LIN {X 0,Y 353.397,Z 547.439,A -85,B 0,C 180,E1 -13404.296,E2 -13404.296} C_VEL
LIN {X 0,Y 353.36,Z 549.314,A -85,B 0,C 180,E1 -13405.439,E2 -13405.439} C_VEL
LIN {X 0,Y 353.319,Z 551.736,A -85,B 0,C 180,E1 -13407.722,E2 -13407.722} C_VEL
LIN {X 0,Y 353.4,Z 552.359,A -85,B 0,C 180,E1 -13408.863,E2 -13408.863} C_VEL
LIN {X 0,Y 353.411,Z 552.568,A -85,B 0,C 180,E1 -13410.002,E2 -13410.002} C_VEL
LIN {X 0,Y 353.421,Z 552.342,A -85,B 0,C 180,E1 -13411.142,E2 -13411.142} C_VEL
LIN {X 0,Y 353.333,Z 551.718,A -85,B 0,C 180,E1 -13412.282,E2 -13412.282} C_VEL
LIN {X 0,Y 353.284,Z 550.703,A -85,B 0,C 180,E1 -13413.424,E2 -13413.424} C_VEL
LIN {X 0,Y 353.361,Z 549.273,A -85,B 0,C 180,E1 -13414.565,E2 -13414.565} C_VEL
LIN {X 0,Y 353.448,Z 546.504,A -85,B 0,C 180,E1 -13416.169,E2 -13416.169} C_VEL
LIN {X 0,Y 353.656,Z 542.242,A -85,B 0,C 180,E1 -13417.998,E2 -13417.998} C_VEL
LIN {X 0,Y 354.205,Z 536.027,A -85,B 0,C 180,E1 -13420,E2 -13420} C_VEL
LIN {X 0,Y 354.806,Z 529.25,A -85,B 0,C 180,E1 -13421.716,E2 -13421.716} C_VEL
LIN {X 0,Y 355.835,Z 520.862,A -85,B 0,C 180,E1 -13423.421,E2 -13423.421} C_VEL
LIN {X 0,Y 356.841,Z 510.928,A -85,B 0,C 180,E1 -13425.028,E2 -13425.028} C_VEL
LIN {X 0,Y 357.899,Z 500.395,A -85,B 0,C 180,E1 -13426.398,E2 -13426.398} C_VEL
LIN {X 0,Y 359.074,Z 489.567,A -85,B 0,C 180,E1 -13427.515,E2 -13427.515} C_VEL
LIN {X 0,Y 359.665,Z 483.015,A -85,B 0,C 180,E1 -13428.073,E2 -13428.073} C_VEL
LIN {X 0,Y 358.36,Z 470.302,A -85,B 0,C 180,E1 -13429.064,E2 -13429.064} C_VEL
LIN {X 0,Y 356.589,Z 457.253,A -85,B 0,C 180,E1 -13429.846,E2 -13429.846} C_VEL
LIN {X 0,Y 354.382,Z 444.691,A -85,B 0,C 180,E1 -13430.404,E2 -13430.404} C_VEL
LIN {X 0,Y 354.887,Z 437.431,A -85,B 0,C 180,E1 -13433.864,E2 -13433.864} C_VEL
LIN {X 0,Y 355.469,Z 430.621,A -85,B 0,C 180,E1 -13437.164,E2 -13437.164} C_VEL
LIN {X 0,Y 356.132,Z 424.489,A -85,B 0,C 180,E1 -13440.223,E2 -13440.223} C_VEL
LIN {X 0,Y 356.859,Z 418.153,A -85,B 0,C 180,E1 -13443.467,E2 -13443.467} C_VEL
LIN {X 0,Y 357.34,Z 414.367,A -85,B 0,C 180,E1 -13445.466,E2 -13445.466} C_VEL
LIN {X 0,Y 357.336,Z 410.539,A -85,B 0,C 180,E1 -13447.57,E2 -13447.57} C_VEL
LIN {X 0,Y 356.459,Z 405.441,A -85,B 0,C 180,E1 -13450.591,E2 -13450.591} C_VEL
LIN {X 0,Y 355.582,Z 400.398,A -85,B 0,C 180,E1 -13453.772,E2 -13453.772} C_VEL
LIN {X 0,Y 354.823,Z 396.289,A -85,B 0,C 180,E1 -13456.533,E2 -13456.533} C_VEL
LIN {X 0,Y 354.822,Z 396.289,A -85,B 0,C 180,E1 -13460.667,E2 -13460.667} C_VEL
LIN {X 0,Y 354.828,Z 396.285,A -85,B 0,C 180,E1 -13464.301,E2 -13464.301} C_VEL
LIN {X 0,Y 354.793,Z 396.287,A -85,B 0,C 180,E1 -13467.667,E2 -13467.667} C_VEL
LIN {X 0,Y 354.853,Z 396.28,A -85,B 0,C 180,E1 -13471.619,E2 -13471.619} C_VEL
LIN {X 0,Y 354.906,Z 396.275,A -85,B 0,C 180,E1 -13474.173,E2 -13474.173} C_VEL
LIN {X 0,Y 354.841,Z 396.282,A -85,B 0,C 180,E1 -13477.894,E2 -13477.894} C_VEL
LIN {X 0,Y 354.929,Z 396.272,A -85,B 0,C 180,E1 -13481.892,E2 -13481.892} C_VEL
LIN {X 0,Y 354.949,Z 396.27,A -85,B 0,C 180,E1 -13485.982,E2 -13485.982} C_VEL
LIN {X 0,Y 354.984,Z 396.265,A -85,B 0,C 180,E1 -13489.736,E2 -13489.736} C_VEL
LIN {X 0,Y 355.13,Z 396.245,A -85,B 0,C 180,E1 -13493.181,E2 -13493.181} C_VEL
LIN {X 0,Y 355.249,Z 396.233,A -85,B 0,C 180,E1 -13497.732,E2 -13497.732} C_VEL
LIN {X 0,Y 355.381,Z 396.22,A -85,B 0,C 180,E1 -13500,E2 -13500} C_VEL
LIN {X 0,Y 355.249,Z 396.235,A -85,B 0,C 180,E1 -13502.268,E2 -13502.268} C_VEL
LIN {X 0,Y 355.143,Z 396.244,A -85,B 0,C 180,E1 -13506.819,E2 -13506.819} C_VEL
LIN {X 0,Y 355.022,Z 396.259,A -85,B 0,C 180,E1 -13509.112,E2 -13509.112} C_VEL
LIN {X 0,Y 354.927,Z 396.271,A -85,B 0,C 180,E1 -13512.581,E2 -13512.581} C_VEL
LIN {X 0,Y 354.896,Z 396.278,A -85,B 0,C 180,E1 -13516.096,E2 -13516.096} C_VEL
LIN {X 0,Y 354.908,Z 396.274,A -85,B 0,C 180,E1 -13518.472,E2 -13518.472} C_VEL
LIN {X 0,Y 354.841,Z 396.283,A -85,B 0,C 180,E1 -13522.106,E2 -13522.106} C_VEL
LIN {X 0,Y 354.905,Z 396.277,A -85,B 0,C 180,E1 -13525.827,E2 -13525.827} C_VEL
LIN {X 0,Y 354.824,Z 396.288,A -85,B 0,C 180,E1 -13529.681,E2 -13529.681} C_VEL
LIN {X 0,Y 354.813,Z 396.288,A -85,B 0,C 180,E1 -13533.701,E2 -13533.701} C_VEL
LIN {X 0,Y 354.803,Z 396.286,A -85,B 0,C 180,E1 -13536.459,E2 -13536.459} C_VEL
LIN {X 0,Y 354.83,Z 396.288,A -85,B 0,C 180,E1 -13539.423,E2 -13539.423} C_VEL
LIN {X 0,Y 354.794,Z 396.29,A -85,B 0,C 180,E1 -13542.866,E2 -13542.866} C_VEL
LIN {X 0,Y 354.786,Z 396.288,A -85,B 0,C 180,E1 -13546.105,E2 -13546.105} C_VEL
LIN {X 0,Y 354.794,Z 396.293,A -85,B 0,C 180,E1 -13549.178,E2 -13549.178} C_VEL
LIN {X 0,Y 354.813,Z 396.286,A -85,B 0,C 180,E1 -13552.401,E2 -13552.401} C_VEL
LIN {X 0,Y 354.818,Z 396.29,A -85,B 0,C 180,E1 -13554.94,E2 -13554.94} C_VEL
LIN {X 0,Y 354.799,Z 396.288,A -85,B 0,C 180,E1 -13558.404,E2 -13558.404} C_VEL
LIN {X 0,Y 354.852,Z 396.281,A -85,B 0,C 180,E1 -13561.617,E2 -13561.617} C_VEL
LIN {X 0,Y 354.905,Z 396.274,A -85,B 0,C 180,E1 -13564.171,E2 -13564.171} C_VEL
LIN {X 0,Y 354.84,Z 396.282,A -85,B 0,C 180,E1 -13567.892,E2 -13567.892} C_VEL
LIN {X 0,Y 354.927,Z 396.271,A -85,B 0,C 180,E1 -13571.89,E2 -13571.89} C_VEL
LIN {X 0,Y 354.932,Z 396.271,A -85,B 0,C 180,E1 -13575.989,E2 -13575.989} C_VEL
LIN {X 0,Y 354.671,Z 396.303,A -85,B 0,C 180,E1 -13579.725,E2 -13579.725} C_VEL
LIN {X 0,Y 354.46,Z 396.335,A -85,B 0,C 180,E1 -13582.02,E2 -13582.02} C_VEL
LIN {X 0,Y 354.473,Z 399.377,A -85,B 0,C 180,E1 -13585.449,E2 -13585.449} C_VEL
LIN {X 0,Y 353.943,Z 403.666,A -85,B 0,C 180,E1 -13589.998,E2 -13589.998} C_VEL
LIN {X 0,Y 354.03,Z 406.198,A -85,B 0,C 180,E1 -13592.771,E2 -13592.771} C_VEL
LIN {X 0,Y 358.141,Z 421.163,A -85,B 0,C 180,E1 -13593.644,E2 -13593.644} C_VEL
LIN {X 0,Y 360.649,Z 432.415,A -85,B 0,C 180,E1 -13594.468,E2 -13594.468} C_VEL
LIN {X 0,Y 360.823,Z 435.833,A -85,B 0,C 180,E1 -13594.731,E2 -13594.731} C_VEL
LIN {X 0,Y 359.959,Z 448.009,A -85,B 0,C 180,E1 -13595.741,E2 -13595.741} C_VEL
LIN {X 0,Y 359.07,Z 457.581,A -85,B 0,C 180,E1 -13596.742,E2 -13596.742} C_VEL
LIN {X 0,Y 358.047,Z 466.663,A -85,B 0,C 180,E1 -13597.895,E2 -13597.895} C_VEL
LIN {X 0,Y 356.935,Z 476.618,A -85,B 0,C 180,E1 -13599.462,E2 -13599.462} C_VEL
LIN {X 0,Y 355.973,Z 484.984,A -85,B 0,C 180,E1 -13601.096,E2 -13601.096} C_VEL
LIN {X 0,Y 355.188,Z 492.159,A -85,B 0,C 180,E1 -13602.859,E2 -13602.859} C_VEL
LIN {X 0,Y 354.426,Z 498.743,A -85,B 0,C 180,E1 -13604.936,E2 -13604.936} C_VEL
LIN {X 0,Y 353.984,Z 503.035,A -85,B 0,C 180,E1 -13606.729,E2 -13606.729} C_VEL
LIN {X 0,Y 353.596,Z 506.211,A -85,B 0,C 180,E1 -13608.54,E2 -13608.54} C_VEL
LIN {X 0,Y 353.329,Z 508.636,A -85,B 0,C 180,E1 -13610.793,E2 -13610.793} C_VEL
LIN {X 0,Y 353.29,Z 509.396,A -85,B 0,C 180,E1 -13612.205,E2 -13612.205} C_VEL
LIN {X 0,Y 353.302,Z 509.483,A -85,B 0,C 180,E1 -13613.788,E2 -13613.788} C_VEL
LIN {X 0,Y 353.448,Z 508.434,A -85,B 0,C 180,E1 -13615.938,E2 -13615.938} C_VEL
LIN {X 0,Y 353.619,Z 507.123,A -85,B 0,C 180,E1 -13617.198,E2 -13617.198} C_VEL
LIN {X 0,Y 354.028,Z 504.148,A -85,B 0,C 180,E1 -13619.136,E2 -13619.136} C_VEL
LIN {X 0,Y 354.494,Z 500.016,A -85,B 0,C 180,E1 -13621.025,E2 -13621.025} C_VEL
LIN {X 0,Y 355.202,Z 494.331,A -85,B 0,C 180,E1 -13622.961,E2 -13622.961} C_VEL
LIN {X 0,Y 356.14,Z 486.878,A -85,B 0,C 180,E1 -13624.906,E2 -13624.906} C_VEL
LIN {X 0,Y 357.147,Z 479.057,A -85,B 0,C 180,E1 -13626.528,E2 -13626.528} C_VEL
LIN {X 0,Y 358.209,Z 469.992,A -85,B 0,C 180,E1 -13628.041,E2 -13628.041} C_VEL
LIN {X 0,Y 359.381,Z 459.402,A -85,B 0,C 180,E1 -13629.458,E2 -13629.458} C_VEL
LIN {X 0,Y 360.469,Z 448.14,A -85,B 0,C 180,E1 -13630.656,E2 -13630.656} C_VEL
LIN {X 0,Y 361.473,Z 436.115,A -85,B 0,C 180,E1 -13631.64,E2 -13631.64} C_VEL
LIN {X 0,Y 359.964,Z 428.14,A -85,B 0,C 180,E1 -13632.29,E2 -13632.29} C_VEL
LIN {X 0,Y 359.337,Z 425.606,A -85,B 0,C 180,E1 -13632.478,E2 -13632.478} C_VEL
LIN {X 0,Y 357.891,Z 422.365,A -85,B 0,C 180,E1 -13632.757,E2 -13632.757} C_VEL
LIN {X 0,Y 353.991,Z 417.862,A -85,B 0,C 180,E1 -13633.242,E2 -13633.242} C_VEL
LIN {X 0,Y 348.982,Z 412.465,A -85,B 0,C 180,E1 -13633.805,E2 -13633.805} C_VEL
LIN {X 0,Y 347.7,Z 410.318,A -85,B 0,C 180,E1 -13633.969,E2 -13633.969} C_VEL
LIN {X 0,Y 346.987,Z 407.79,A -85,B 0,C 180,E1 -13634.13,E2 -13634.13} C_VEL
LIN {X 0,Y 347.06,Z 405.464,A -85,B 0,C 180,E1 -13636.798,E2 -13636.798} C_VEL
LIN {X 0,Y 347.154,Z 402.495,A -85,B 0,C 180,E1 -13640.286,E2 -13640.286} C_VEL
LIN {X 0,Y 347.282,Z 400.542,A -85,B 0,C 180,E1 -13642.619,E2 -13642.619} C_VEL
LIN {X 0,Y 347.414,Z 397.753,A -85,B 0,C 180,E1 -13646.032,E2 -13646.032} C_VEL
LIN {X 0,Y 347.48,Z 397.209,A -85,B 0,C 180,E1 -13646.901,E2 -13646.901} C_VEL
LIN {X 0,Y 347.703,Z 397.178,A -85,B 0,C 180,E1 -13649.648,E2 -13649.648} C_VEL
LIN {X 0,Y 347.832,Z 397.16,A -85,B 0,C 180,E1 -13652.744,E2 -13652.744} C_VEL
LIN {X 0,Y 347.8,Z 397.164,A -85,B 0,C 180,E1 -13656.163,E2 -13656.163} C_VEL
LIN {X 0,Y 347.825,Z 397.157,A -85,B 0,C 180,E1 -13659.91,E2 -13659.91} C_VEL
LIN {X 0,Y 347.848,Z 397.156,A -85,B 0,C 180,E1 -13662.358,E2 -13662.358} C_VEL
LIN {X 0,Y 347.878,Z 397.153,A -85,B 0,C 180,E1 -13665.97,E2 -13665.97} C_VEL
LIN {X 0,Y 347.914,Z 397.146,A -85,B 0,C 180,E1 -13669.525,E2 -13669.525} C_VEL
LIN {X 0,Y 348.055,Z 397.13,A -85,B 0,C 180,E1 -13671.874,E2 -13671.874} C_VEL
LIN {X 0,Y 348.053,Z 397.132,A -85,B 0,C 180,E1 -13674.206,E2 -13674.206} C_VEL
LIN {X 0,Y 348.19,Z 397.114,A -85,B 0,C 180,E1 -13677.687,E2 -13677.687} C_VEL
LIN {X 0,Y 348.349,Z 397.094,A -85,B 0,C 180,E1 -13680,E2 -13680} C_VEL
LIN {X 0,Y 348.197,Z 397.113,A -85,B 0,C 180,E1 -13682.314,E2 -13682.314} C_VEL
LIN {X 0,Y 348.086,Z 397.127,A -85,B 0,C 180,E1 -13686.958,E2 -13686.958} C_VEL
LIN {X 0,Y 347.95,Z 397.144,A -85,B 0,C 180,E1 -13689.299,E2 -13689.299} C_VEL
LIN {X 0,Y 347.874,Z 397.154,A -85,B 0,C 180,E1 -13692.84,E2 -13692.84} C_VEL
LIN {X 0,Y 347.821,Z 397.16,A -85,B 0,C 180,E1 -13696.432,E2 -13696.432} C_VEL
LIN {X 0,Y 347.845,Z 397.157,A -85,B 0,C 180,E1 -13698.861,E2 -13698.861} C_VEL
LIN {X 0,Y 347.823,Z 397.164,A -85,B 0,C 180,E1 -13702.576,E2 -13702.576} C_VEL
LIN {X 0,Y 347.815,Z 397.165,A -85,B 0,C 180,E1 -13706.394,E2 -13706.394} C_VEL
LIN {X 0,Y 347.733,Z 397.174,A -85,B 0,C 180,E1 -13710.35,E2 -13710.35} C_VEL
LIN {X 0,Y 347.733,Z 397.172,A -85,B 0,C 180,E1 -13714.046,E2 -13714.046} C_VEL
LIN {X 0,Y 347.749,Z 397.171,A -85,B 0,C 180,E1 -13717.323,E2 -13717.323} C_VEL
LIN {X 0,Y 347.78,Z 397.17,A -85,B 0,C 180,E1 -13720.291,E2 -13720.291} C_VEL
LIN {X 0,Y 347.785,Z 397.199,A -85,B 0,C 180,E1 -13722.215,E2 -13722.215} C_VEL
LIN {X 0,Y 348.524,Z 400.99,A -85,B 0,C 180,E1 -13725.112,E2 -13725.112} C_VEL
LIN {X 0,Y 349.547,Z 406.827,A -85,B 0,C 180,E1 -13729.167,E2 -13729.167} C_VEL
LIN {X 0,Y 350.336,Z 411.714,A -85,B 0,C 180,E1 -13732.28,E2 -13732.28} C_VEL
LIN {X 0,Y 350.474,Z 413.477,A -85,B 0,C 180,E1 -13733.333,E2 -13733.333} C_VEL
LIN {X 0,Y 350.004,Z 417.843,A -85,B 0,C 180,E1 -13735.793,E2 -13735.793} C_VEL
LIN {X 0,Y 349.083,Z 425.275,A -85,B 0,C 180,E1 -13739.783,E2 -13739.783} C_VEL
LIN {X 0,Y 348.248,Z 432.816,A -85,B 0,C 180,E1 -13743.645,E2 -13743.645} C_VEL
LIN {X 0,Y 347.565,Z 440.422,A -85,B 0,C 180,E1 -13747.409,E2 -13747.409} C_VEL
LIN {X 0,Y 347.348,Z 443.506,A -85,B 0,C 180,E1 -13748.917,E2 -13748.917} C_VEL
LIN {X 0,Y 349.982,Z 457.043,A -85,B 0,C 180,E1 -13749.582,E2 -13749.582} C_VEL
LIN {X 0,Y 351.593,Z 469.541,A -85,B 0,C 180,E1 -13750.376,E2 -13750.376} C_VEL
LIN {X 0,Y 352.839,Z 482.403,A -85,B 0,C 180,E1 -13751.419,E2 -13751.419} C_VEL
LIN {X 0,Y 352.669,Z 487.333,A -85,B 0,C 180,E1 -13751.861,E2 -13751.861} C_VEL
LIN {X 0,Y 351.401,Z 498.465,A -85,B 0,C 180,E1 -13752.995,E2 -13752.995} C_VEL
LIN {X 0,Y 350.256,Z 508.181,A -85,B 0,C 180,E1 -13754.236,E2 -13754.236} C_VEL
LIN {X 0,Y 349.213,Z 517.642,A -85,B 0,C 180,E1 -13755.73,E2 -13755.73} C_VEL
LIN {X 0,Y 348.167,Z 526.574,A -85,B 0,C 180,E1 -13757.47,E2 -13757.47} C_VEL
LIN {X 0,Y 347.381,Z 533.764,A -85,B 0,C 180,E1 -13759.217,E2 -13759.217} C_VEL
LIN {X 0,Y 346.733,Z 540.34,A -85,B 0,C 180,E1 -13761.259,E2 -13761.259} C_VEL
LIN {X 0,Y 346.437,Z 544.705,A -85,B 0,C 180,E1 -13763.011,E2 -13763.011} C_VEL
LIN {X 0,Y 346.337,Z 547.027,A -85,B 0,C 180,E1 -13764.179,E2 -13764.179} C_VEL
LIN {X 0,Y 346.274,Z 548.895,A -85,B 0,C 180,E1 -13765.346,E2 -13765.346} C_VEL
LIN {X 0,Y 346.224,Z 551.312,A -85,B 0,C 180,E1 -13767.676,E2 -13767.676} C_VEL
LIN {X 0,Y 346.321,Z 551.933,A -85,B 0,C 180,E1 -13768.839,E2 -13768.839} C_VEL
LIN {X 0,Y 346.35,Z 552.137,A -85,B 0,C 180,E1 -13770.002,E2 -13770.002} C_VEL
LIN {X 0,Y 346.34,Z 551.906,A -85,B 0,C 180,E1 -13771.165,E2 -13771.165} C_VEL
LIN {X 0,Y 346.207,Z 550.26,A -85,B 0,C 180,E1 -13773.494,E2 -13773.494} C_VEL
LIN {X 0,Y 346.275,Z 548.823,A -85,B 0,C 180,E1 -13774.659,E2 -13774.659} C_VEL
LIN {X 0,Y 346.345,Z 546.379,A -85,B 0,C 180,E1 -13776.117,E2 -13776.117} C_VEL
LIN {X 0,Y 346.594,Z 541.777,A -85,B 0,C 180,E1 -13778.162,E2 -13778.162} C_VEL
LIN {X 0,Y 347.174,Z 535.549,A -85,B 0,C 180,E1 -13780.205,E2 -13780.205} C_VEL
LIN {X 0,Y 347.818,Z 528.762,A -85,B 0,C 180,E1 -13781.955,E2 -13781.955} C_VEL
LIN {X 0,Y 348.859,Z 520.356,A -85,B 0,C 180,E1 -13783.695,E2 -13783.695} C_VEL
LIN {X 0,Y 349.897,Z 510.606,A -85,B 0,C 180,E1 -13785.303,E2 -13785.303} C_VEL
LIN {X 0,Y 351.08,Z 499.852,A -85,B 0,C 180,E1 -13786.726,E2 -13786.726} C_VEL
LIN {X 0,Y 352.28,Z 488.975,A -85,B 0,C 180,E1 -13787.864,E2 -13787.864} C_VEL
LIN {X 0,Y 352.66,Z 482.378,A -85,B 0,C 180,E1 -13788.445,E2 -13788.445} C_VEL
LIN {X 0,Y 351.429,Z 470.426,A -85,B 0,C 180,E1 -13789.398,E2 -13789.398} C_VEL
LIN {X 0,Y 349.705,Z 457.486,A -85,B 0,C 180,E1 -13790.204,E2 -13790.204} C_VEL
LIN {X 0,Y 347.371,Z 444.293,A -85,B 0,C 180,E1 -13790.815,E2 -13790.815} C_VEL
LIN {X 0,Y 347.93,Z 436.473,A -85,B 0,C 180,E1 -13794.635,E2 -13794.635} C_VEL
LIN {X 0,Y 348.646,Z 429.181,A -85,B 0,C 180,E1 -13798.277,E2 -13798.277} C_VEL
LIN {X 0,Y 349.334,Z 422.844,A -85,B 0,C 180,E1 -13801.541,E2 -13801.541} C_VEL
LIN {X 0,Y 350.155,Z 417.016,A -85,B 0,C 180,E1 -13804.622,E2 -13804.622} C_VEL
LIN {X 0,Y 350.457,Z 412.746,A -85,B 0,C 180,E1 -13806.987,E2 -13806.987} C_VEL
LIN {X 0,Y 349.634,Z 407.634,A -85,B 0,C 180,E1 -13810.035,E2 -13810.035} C_VEL
LIN {X 0,Y 348.707,Z 402.209,A -85,B 0,C 180,E1 -13813.484,E2 -13813.484} C_VEL
LIN {X 0,Y 347.757,Z 397.17,A -85,B 0,C 180,E1 -13816.974,E2 -13816.974} C_VEL
LIN {X 0,Y 347.754,Z 397.168,A -85,B 0,C 180,E1 -13820.174,E2 -13820.174} C_VEL
LIN {X 0,Y 347.768,Z 397.168,A -85,B 0,C 180,E1 -13822.68,E2 -13822.68} C_VEL
LIN {X 0,Y 347.755,Z 397.164,A -85,B 0,C 180,E1 -13825.957,E2 -13825.957} C_VEL
LIN {X 0,Y 347.756,Z 397.164,A -85,B 0,C 180,E1 -13829.653,E2 -13829.653} C_VEL
LIN {X 0,Y 347.838,Z 397.154,A -85,B 0,C 180,E1 -13833.608,E2 -13833.608} C_VEL
LIN {X 0,Y 347.796,Z 397.161,A -85,B 0,C 180,E1 -13836.162,E2 -13836.162} C_VEL
LIN {X 0,Y 347.819,Z 397.157,A -85,B 0,C 180,E1 -13839.91,E2 -13839.91} C_VEL
LIN {X 0,Y 347.873,Z 397.155,A -85,B 0,C 180,E1 -13842.359,E2 -13842.359} C_VEL
LIN {X 0,Y 347.905,Z 397.148,A -85,B 0,C 180,E1 -13845.971,E2 -13845.971} C_VEL
LIN {X 0,Y 347.935,Z 397.142,A -85,B 0,C 180,E1 -13849.526,E2 -13849.526} C_VEL
LIN {X 0,Y 348.097,Z 397.122,A -85,B 0,C 180,E1 -13853.042,E2 -13853.042} C_VEL
LIN {X 0,Y 348.211,Z 397.109,A -85,B 0,C 180,E1 -13857.686,E2 -13857.686} C_VEL
LIN {X 0,Y 348.331,Z 397.098,A -85,B 0,C 180,E1 -13860,E2 -13860} C_VEL
LIN {X 0,Y 348.211,Z 397.11,A -85,B 0,C 180,E1 -13862.313,E2 -13862.313} C_VEL
LIN {X 0,Y 348.111,Z 397.12,A -85,B 0,C 180,E1 -13866.957,E2 -13866.957} C_VEL
LIN {X 0,Y 347.935,Z 397.143,A -85,B 0,C 180,E1 -13870.474,E2 -13870.474} C_VEL
LIN {X 0,Y 347.905,Z 397.148,A -85,B 0,C 180,E1 -13874.15,E2 -13874.15} C_VEL
LIN {X 0,Y 347.897,Z 397.147,A -85,B 0,C 180,E1 -13878.29,E2 -13878.29} C_VEL
LIN {X 0,Y 347.795,Z 397.165,A -85,B 0,C 180,E1 -13881.634,E2 -13881.634} C_VEL
LIN {X 0,Y 347.819,Z 397.158,A -85,B 0,C 180,E1 -13885.108,E2 -13885.108} C_VEL
LIN {X 0,Y 347.815,Z 397.161,A -85,B 0,C 180,E1 -13887.693,E2 -13887.693} C_VEL
LIN {X 0,Y 347.755,Z 397.164,A -85,B 0,C 180,E1 -13890.347,E2 -13890.347} C_VEL
LIN {X 0,Y 347.755,Z 397.165,A -85,B 0,C 180,E1 -13894.043,E2 -13894.043} C_VEL
LIN {X 0,Y 347.767,Z 397.168,A -85,B 0,C 180,E1 -13897.32,E2 -13897.32} C_VEL
LIN {X 0,Y 347.738,Z 397.166,A -85,B 0,C 180,E1 -13900.296,E2 -13900.296} C_VEL
LIN {X 0,Y 347.729,Z 397.171,A -85,B 0,C 180,E1 -13903.407,E2 -13903.407} C_VEL
LIN {X 0,Y 347.734,Z 397.168,A -85,B 0,C 180,E1 -13906.685,E2 -13906.685} C_VEL
LIN {X 0,Y 347.753,Z 397.164,A -85,B 0,C 180,E1 -13910.172,E2 -13910.172} C_VEL
LIN {X 0,Y 347.768,Z 397.165,A -85,B 0,C 180,E1 -13912.678,E2 -13912.678} C_VEL
LIN {X 0,Y 347.754,Z 397.164,A -85,B 0,C 180,E1 -13915.955,E2 -13915.955} C_VEL
LIN {X 0,Y 347.755,Z 397.164,A -85,B 0,C 180,E1 -13919.651,E2 -13919.651} C_VEL
LIN {X 0,Y 347.836,Z 397.154,A -85,B 0,C 180,E1 -13923.606,E2 -13923.606} C_VEL
LIN {X 0,Y 347.794,Z 397.16,A -85,B 0,C 180,E1 -13926.16,E2 -13926.16} C_VEL
LIN {X 0,Y 347.817,Z 397.156,A -85,B 0,C 180,E1 -13929.908,E2 -13929.908} C_VEL
LIN {X 0,Y 347.871,Z 397.152,A -85,B 0,C 180,E1 -13932.358,E2 -13932.358} C_VEL
LIN {X 0,Y 347.901,Z 397.147,A -85,B 0,C 180,E1 -13935.969,E2 -13935.969} C_VEL
LIN {X 0,Y 347.657,Z 397.176,A -85,B 0,C 180,E1 -13939.515,E2 -13939.515} C_VEL
LIN {X 0,Y 347.434,Z 397.208,A -85,B 0,C 180,E1 -13941.858,E2 -13941.858} C_VEL
LIN {X 0,Y 347.44,Z 400.136,A -85,B 0,C 180,E1 -13945.357,E2 -13945.357} C_VEL
LIN {X 0,Y 346.885,Z 404.449,A -85,B 0,C 180,E1 -13949.998,E2 -13949.998} C_VEL
LIN {X 0,Y 346.935,Z 406.636,A -85,B 0,C 180,E1 -13952.356,E2 -13952.356} C_VEL
LIN {X 0,Y 351.006,Z 420.997,A -85,B 0,C 180,E1 -13953.226,E2 -13953.226} C_VEL
LIN {X 0,Y 353.758,Z 433.144,A -85,B 0,C 180,E1 -13954.135,E2 -13954.135} C_VEL
LIN {X 0,Y 354.051,Z 436.48,A -85,B 0,C 180,E1 -13954.405,E2 -13954.405} C_VEL
LIN {X 0,Y 353.176,Z 448.27,A -85,B 0,C 180,E1 -13955.4,E2 -13955.4} C_VEL
LIN {X 0,Y 352.234,Z 458.052,A -85,B 0,C 180,E1 -13956.442,E2 -13956.442} C_VEL
LIN {X 0,Y 351.079,Z 468.119,A -85,B 0,C 180,E1 -13957.763,E2 -13957.763} C_VEL
LIN {X 0,Y 350.004,Z 477.238,A -85,B 0,C 180,E1 -13959.242,E2 -13959.242} C_VEL
LIN {X 0,Y 349.113,Z 484.74,A -85,B 0,C 180,E1 -13960.729,E2 -13960.729} C_VEL
LIN {X 0,Y 348.247,Z 492.091,A -85,B 0,C 180,E1 -13962.527,E2 -13962.527} C_VEL
LIN {X 0,Y 347.632,Z 497.065,A -85,B 0,C 180,E1 -13964.038,E2 -13964.038} C_VEL
LIN {X 0,Y 347.116,Z 501.841,A -85,B 0,C 180,E1 -13965.86,E2 -13965.86} C_VEL
LIN {X 0,Y 346.685,Z 505.459,A -85,B 0,C 180,E1 -13967.7,E2 -13967.7} C_VEL
LIN {X 0,Y 346.46,Z 507.25,A -85,B 0,C 180,E1 -13968.936,E2 -13968.936} C_VEL
LIN {X 0,Y 346.253,Z 509.224,A -85,B 0,C 180,E1 -13970.985,E2 -13970.985} C_VEL
LIN {X 0,Y 346.185,Z 509.916,A -85,B 0,C 180,E1 -13972.686,E2 -13972.686} C_VEL
LIN {X 0,Y 346.227,Z 509.896,A -85,B 0,C 180,E1 -13974.014,E2 -13974.014} C_VEL
LIN {X 0,Y 346.273,Z 509.403,A -85,B 0,C 180,E1 -13975.225,E2 -13975.225} C_VEL
LIN {X 0,Y 346.488,Z 508.125,A -85,B 0,C 180,E1 -13976.814,E2 -13976.814} C_VEL
LIN {X 0,Y 346.794,Z 506.003,A -85,B 0,C 180,E1 -13978.437,E2 -13978.437} C_VEL
LIN {X 0,Y 347.23,Z 502.364,A -85,B 0,C 180,E1 -13980.395,E2 -13980.395} C_VEL
LIN {X 0,Y 347.922,Z 497.176,A -85,B 0,C 180,E1 -13982.407,E2 -13982.407} C_VEL
LIN {X 0,Y 348.827,Z 490.635,A -85,B 0,C 180,E1 -13984.338,E2 -13984.338} C_VEL
LIN {X 0,Y 349.7,Z 483.775,A -85,B 0,C 180,E1 -13985.956,E2 -13985.956} C_VEL
LIN {X 0,Y 350.874,Z 474.829,A -85,B 0,C 180,E1 -13987.652,E2 -13987.652} C_VEL
LIN {X 0,Y 352.049,Z 464.804,A -85,B 0,C 180,E1 -13989.166,E2 -13989.166} C_VEL
LIN {X 0,Y 353.255,Z 454.028,A -85,B 0,C 180,E1 -13990.468,E2 -13990.468} C_VEL
LIN {X 0,Y 354.332,Z 442.706,A -85,B 0,C 180,E1 -13991.541,E2 -13991.541} C_VEL
LIN {X 0,Y 354.748,Z 436.625,A -85,B 0,C 180,E1 -13992.021,E2 -13992.021} C_VEL
LIN {X 0,Y 352.006,Z 424.655,A -85,B 0,C 180,E1 -13993.01,E2 -13993.01} C_VEL
LIN {X 0,Y 348.401,Z 412.41,A -85,B 0,C 180,E1 -13993.847,E2 -13993.847} C_VEL
LIN {X 0,Y 347.7,Z 410.318,A -85,B 0,C 180,E1 -13993.969,E2 -13993.969} C_VEL
LIN {X 0,Y 346.554,Z 408.686,A -85,B 0,C 180,E1 -13994.208,E2 -13994.208} C_VEL
LIN {X 0,Y 344.636,Z 407.492,A -85,B 0,C 180,E1 -13994.816,E2 -13994.816} C_VEL
LIN {X 0,Y 342.19,Z 406.75,A -85,B 0,C 180,E1 -13996.035,E2 -13996.035} C_VEL
LIN {X 0,Y 340.594,Z 405.909,A -85,B 0,C 180,E1 -13997.496,E2 -13997.496} C_VEL
LIN {X 0,Y 340.059,Z 404.553,A -85,B 0,C 180,E1 -13998.976,E2 -13998.976} C_VEL
LIN {X 0,Y 340.227,Z 402.274,A -85,B 0,C 180,E1 -14001.712,E2 -14001.712} C_VEL
LIN {X 0,Y 340.321,Z 399.878,A -85,B 0,C 180,E1 -14004.674,E2 -14004.674} C_VEL
LIN {X 0,Y 340.392,Z 398.73,A -85,B 0,C 180,E1 -14006.119,E2 -14006.119} C_VEL
LIN {X 0,Y 340.539,Z 398.074,A -85,B 0,C 180,E1 -14007.789,E2 -14007.789} C_VEL
LIN {X 0,Y 340.709,Z 398.047,A -85,B 0,C 180,E1 -14010.326,E2 -14010.326} C_VEL
LIN {X 0,Y 340.786,Z 398.037,A -85,B 0,C 180,E1 -14013.018,E2 -14013.018} C_VEL
LIN {X 0,Y 340.774,Z 398.04,A -85,B 0,C 180,E1 -14016.93,E2 -14016.93} C_VEL
LIN {X 0,Y 340.788,Z 398.037,A -85,B 0,C 180,E1 -14020.733,E2 -14020.733} C_VEL
LIN {X 0,Y 340.768,Z 398.04,A -85,B 0,C 180,E1 -14023.218,E2 -14023.218} C_VEL
LIN {X 0,Y 340.828,Z 398.028,A -85,B 0,C 180,E1 -14026.89,E2 -14026.89} C_VEL
LIN {X 0,Y 340.911,Z 398.019,A -85,B 0,C 180,E1 -14030.507,E2 -14030.507} C_VEL
LIN {X 0,Y 341.059,Z 397.998,A -85,B 0,C 180,E1 -14032.898,E2 -14032.898} C_VEL
LIN {X 0,Y 341.152,Z 397.99,A -85,B 0,C 180,E1 -14037.639,E2 -14037.639} C_VEL
LIN {X 0,Y 341.298,Z 397.972,A -85,B 0,C 180,E1 -14040,E2 -14040} C_VEL
LIN {X 0,Y 341.159,Z 397.99,A -85,B 0,C 180,E1 -14042.361,E2 -14042.361} C_VEL
LIN {X 0,Y 341.056,Z 398.003,A -85,B 0,C 180,E1 -14047.102,E2 -14047.102} C_VEL
LIN {X 0,Y 340.856,Z 398.026,A -85,B 0,C 180,E1 -14050.694,E2 -14050.694} C_VEL
LIN {X 0,Y 340.844,Z 398.029,A -85,B 0,C 180,E1 -14054.326,E2 -14054.326} C_VEL
LIN {X 0,Y 340.821,Z 398.033,A -85,B 0,C 180,E1 -14058.469,E2 -14058.469} C_VEL
LIN {X 0,Y 340.795,Z 398.037,A -85,B 0,C 180,E1 -14061.883,E2 -14061.883} C_VEL
LIN {X 0,Y 340.76,Z 398.043,A -85,B 0,C 180,E1 -14065.666,E2 -14065.666} C_VEL
LIN {X 0,Y 340.712,Z 398.049,A -85,B 0,C 180,E1 -14068.322,E2 -14068.322} C_VEL
LIN {X 0,Y 340.682,Z 398.052,A -85,B 0,C 180,E1 -14071.047,E2 -14071.047} C_VEL
LIN {X 0,Y 340.704,Z 398.048,A -85,B 0,C 180,E1 -14075.281,E2 -14075.281} C_VEL
LIN {X 0,Y 340.704,Z 398.049,A -85,B 0,C 180,E1 -14078.39,E2 -14078.39} C_VEL
LIN {X 0,Y 340.752,Z 398.118,A -85,B 0,C 180,E1 -14081.689,E2 -14081.689} C_VEL
LIN {X 0,Y 341.417,Z 401.553,A -85,B 0,C 180,E1 -14084.418,E2 -14084.418} C_VEL
LIN {X 0,Y 342.163,Z 406.035,A -85,B 0,C 180,E1 -14087.684,E2 -14087.684} C_VEL
LIN {X 0,Y 343.07,Z 411.152,A -85,B 0,C 180,E1 -14091.12,E2 -14091.12} C_VEL
LIN {X 0,Y 343.439,Z 415.151,A -85,B 0,C 180,E1 -14093.602,E2 -14093.602} C_VEL
LIN {X 0,Y 342.834,Z 420.066,A -85,B 0,C 180,E1 -14096.397,E2 -14096.397} C_VEL
LIN {X 0,Y 341.85,Z 427.473,A -85,B 0,C 180,E1 -14100.438,E2 -14100.438} C_VEL
LIN {X 0,Y 341.045,Z 434.974,A -85,B 0,C 180,E1 -14104.361,E2 -14104.361} C_VEL
LIN {X 0,Y 340.345,Z 443.121,A -85,B 0,C 180,E1 -14108.437,E2 -14108.437} C_VEL
LIN {X 0,Y 343.055,Z 456.588,A -85,B 0,C 180,E1 -14109.124,E2 -14109.124} C_VEL
LIN {X 0,Y 344.721,Z 469.437,A -85,B 0,C 180,E1 -14109.97,E2 -14109.97} C_VEL
LIN {X 0,Y 345.88,Z 482.178,A -85,B 0,C 180,E1 -14111.031,E2 -14111.031} C_VEL
LIN {X 0,Y 345.929,Z 487.092,A -85,B 0,C 180,E1 -14111.494,E2 -14111.494} C_VEL
LIN {X 0,Y 344.572,Z 498.178,A -85,B 0,C 180,E1 -14112.647,E2 -14112.647} C_VEL
LIN {X 0,Y 343.349,Z 508.192,A -85,B 0,C 180,E1 -14113.962,E2 -14113.962} C_VEL
LIN {X 0,Y 342.314,Z 517.302,A -85,B 0,C 180,E1 -14115.436,E2 -14115.436} C_VEL
LIN {X 0,Y 341.183,Z 526.217,A -85,B 0,C 180,E1 -14117.209,E2 -14117.209} C_VEL
LIN {X 0,Y 340.342,Z 533.386,A -85,B 0,C 180,E1 -14118.991,E2 -14118.991} C_VEL
LIN {X 0,Y 339.696,Z 539.951,A -85,B 0,C 180,E1 -14121.076,E2 -14121.076} C_VEL
LIN {X 0,Y 339.363,Z 544.303,A -85,B 0,C 180,E1 -14122.865,E2 -14122.865} C_VEL
LIN {X 0,Y 339.257,Z 546.62,A -85,B 0,C 180,E1 -14124.057,E2 -14124.057} C_VEL
LIN {X 0,Y 339.193,Z 548.479,A -85,B 0,C 180,E1 -14125.248,E2 -14125.248} C_VEL
LIN {X 0,Y 339.13,Z 550.888,A -85,B 0,C 180,E1 -14127.627,E2 -14127.627} C_VEL
LIN {X 0,Y 339.227,Z 551.506,A -85,B 0,C 180,E1 -14128.815,E2 -14128.815} C_VEL
LIN {X 0,Y 339.29,Z 551.705,A -85,B 0,C 180,E1 -14130.002,E2 -14130.002} C_VEL
LIN {X 0,Y 339.26,Z 551.471,A -85,B 0,C 180,E1 -14131.189,E2 -14131.189} C_VEL
LIN {X 0,Y 339.132,Z 549.817,A -85,B 0,C 180,E1 -14133.567,E2 -14133.567} C_VEL
LIN {X 0,Y 339.194,Z 548.371,A -85,B 0,C 180,E1 -14134.756,E2 -14134.756} C_VEL
LIN {X 0,Y 339.3,Z 545.37,A -85,B 0,C 180,E1 -14136.543,E2 -14136.543} C_VEL
LIN {X 0,Y 339.549,Z 541.306,A -85,B 0,C 180,E1 -14138.333,E2 -14138.333} C_VEL
LIN {X 0,Y 340.146,Z 535.061,A -85,B 0,C 180,E1 -14140.418,E2 -14140.418} C_VEL
LIN {X 0,Y 340.848,Z 528.258,A -85,B 0,C 180,E1 -14142.203,E2 -14142.203} C_VEL
LIN {X 0,Y 341.89,Z 519.822,A -85,B 0,C 180,E1 -14143.979,E2 -14143.979} C_VEL
LIN {X 0,Y 342.894,Z 511.129,A -85,B 0,C 180,E1 -14145.455,E2 -14145.455} C_VEL
LIN {X 0,Y 344.107,Z 500.438,A -85,B 0,C 180,E1 -14146.922,E2 -14146.922} C_VEL
LIN {X 0,Y 345.333,Z 489.847,A -85,B 0,C 180,E1 -14148.083,E2 -14148.083} C_VEL
LIN {X 0,Y 345.78,Z 483.476,A -85,B 0,C 180,E1 -14148.672,E2 -14148.672} C_VEL
LIN {X 0,Y 344.506,Z 470.63,A -85,B 0,C 180,E1 -14149.738,E2 -14149.738} C_VEL
LIN {X 0,Y 342.772,Z 457.349,A -85,B 0,C 180,E1 -14150.595,E2 -14150.595} C_VEL
LIN {X 0,Y 340.358,Z 443.875,A -85,B 0,C 180,E1 -14151.242,E2 -14151.242} C_VEL
LIN {X 0,Y 340.899,Z 436.614,A -85,B 0,C 180,E1 -14154.891,E2 -14154.891} C_VEL
LIN {X 0,Y 341.569,Z 430.051,A -85,B 0,C 180,E1 -14158.247,E2 -14158.247} C_VEL
LIN {X 0,Y 342.291,Z 423.742,A -85,B 0,C 180,E1 -14161.574,E2 -14161.574} C_VEL
LIN {X 0,Y 343.208,Z 417.41,A -85,B 0,C 180,E1 -14165.005,E2 -14165.005} C_VEL
LIN {X 0,Y 343.46,Z 413.787,A -85,B 0,C 180,E1 -14167.057,E2 -14167.057} C_VEL
LIN {X 0,Y 342.491,Z 408.008,A -85,B 0,C 180,E1 -14170.602,E2 -14170.602} C_VEL
LIN {X 0,Y 341.62,Z 402.89,A -85,B 0,C 180,E1 -14173.942,E2 -14173.942} C_VEL
LIN {X 0,Y 340.724,Z 398.045,A -85,B 0,C 180,E1 -14177.342,E2 -14177.342} C_VEL
LIN {X 0,Y 340.706,Z 398.046,A -85,B 0,C 180,E1 -14180.248,E2 -14180.248} C_VEL
LIN {X 0,Y 340.717,Z 398.041,A -85,B 0,C 180,E1 -14183.56,E2 -14183.56} C_VEL
LIN {X 0,Y 340.699,Z 398.044,A -85,B 0,C 180,E1 -14186.154,E2 -14186.154} C_VEL
LIN {X 0,Y 340.748,Z 398.039,A -85,B 0,C 180,E1 -14190.33,E2 -14190.33} C_VEL
LIN {X 0,Y 340.81,Z 398.031,A -85,B 0,C 180,E1 -14193.02,E2 -14193.02} C_VEL
LIN {X 0,Y 340.763,Z 398.035,A -85,B 0,C 180,E1 -14195.639,E2 -14195.639} C_VEL
LIN {X 0,Y 340.752,Z 398.036,A -85,B 0,C 180,E1 -14199.474,E2 -14199.474} C_VEL
LIN {X 0,Y 340.865,Z 398.024,A -85,B 0,C 180,E1 -14201.984,E2 -14201.984} C_VEL
LIN {X 0,Y 340.877,Z 398.021,A -85,B 0,C 180,E1 -14205.705,E2 -14205.705} C_VEL
LIN {X 0,Y 340.877,Z 398.021,A -85,B 0,C 180,E1 -14209.306,E2 -14209.306} C_VEL
LIN {X 0,Y 341.065,Z 397.998,A -85,B 0,C 180,E1 -14212.898,E2 -14212.898} C_VEL
LIN {X 0,Y 341.173,Z 397.985,A -85,B 0,C 180,E1 -14217.639,E2 -14217.639} C_VEL
LIN {X 0,Y 341.282,Z 397.975,A -85,B 0,C 180,E1 -14220,E2 -14220} C_VEL
LIN {X 0,Y 341.173,Z 397.986,A -85,B 0,C 180,E1 -14222.361,E2 -14222.361} C_VEL
LIN {X 0,Y 341.081,Z 397.995,A -85,B 0,C 180,E1 -14227.102,E2 -14227.102} C_VEL
LIN {X 0,Y 340.877,Z 398.021,A -85,B 0,C 180,E1 -14230.694,E2 -14230.694} C_VEL
LIN {X 0,Y 340.87,Z 398.023,A -85,B 0,C 180,E1 -14234.324,E2 -14234.324} C_VEL
LIN {X 0,Y 340.844,Z 398.025,A -85,B 0,C 180,E1 -14238.466,E2 -14238.466} C_VEL
LIN {X 0,Y 340.761,Z 398.039,A -85,B 0,C 180,E1 -14241.856,E2 -14241.856} C_VEL
LIN {X 0,Y 340.779,Z 398.038,A -85,B 0,C 180,E1 -14245.664,E2 -14245.664} C_VEL
LIN {X 0,Y 340.735,Z 398.039,A -85,B 0,C 180,E1 -14248.32,E2 -14248.32} C_VEL
LIN {X 0,Y 340.704,Z 398.044,A -85,B 0,C 180,E1 -14251.044,E2 -14251.044} C_VEL
LIN {X 0,Y 340.724,Z 398.044,A -85,B 0,C 180,E1 -14255.278,E2 -14255.278} C_VEL
LIN {X 0,Y 340.716,Z 398.041,A -85,B 0,C 180,E1 -14258.385,E2 -14258.385} C_VEL
LIN {X 0,Y 340.705,Z 398.042,A -85,B 0,C 180,E1 -14262.044,E2 -14262.044} C_VEL
LIN {X 0,Y 340.69,Z 398.047,A -85,B 0,C 180,E1 -14265.46,E2 -14265.46} C_VEL
LIN {X 0,Y 340.692,Z 398.046,A -85,B 0,C 180,E1 -14268.689,E2 -14268.689} C_VEL
LIN {X 0,Y 340.739,Z 398.038,A -85,B 0,C 180,E1 -14271.771,E2 -14271.771} C_VEL
LIN {X 0,Y 340.729,Z 398.04,A -85,B 0,C 180,E1 -14275.594,E2 -14275.594} C_VEL
LIN {X 0,Y 340.703,Z 398.048,A -85,B 0,C 180,E1 -14278.954,E2 -14278.954} C_VEL
LIN {X 0,Y 340.809,Z 398.034,A -85,B 0,C 180,E1 -14283.018,E2 -14283.018} C_VEL
LIN {X 0,Y 340.761,Z 398.035,A -85,B 0,C 180,E1 -14285.637,E2 -14285.637} C_VEL
LIN {X 0,Y 340.757,Z 398.036,A -85,B 0,C 180,E1 -14289.473,E2 -14289.473} C_VEL
LIN {X 0,Y 340.862,Z 398.023,A -85,B 0,C 180,E1 -14291.982,E2 -14291.982} C_VEL
LIN {X 0,Y 340.856,Z 398.023,A -85,B 0,C 180,E1 -14295.715,E2 -14295.715} C_VEL
LIN {X 0,Y 340.635,Z 398.051,A -85,B 0,C 180,E1 -14299.297,E2 -14299.297} C_VEL
LIN {X 0,Y 340.416,Z 398.081,A -85,B 0,C 180,E1 -14301.689,E2 -14301.689} C_VEL
LIN {X 0,Y 340.365,Z 399.874,A -85,B 0,C 180,E1 -14304.072,E2 -14304.072} C_VEL
LIN {X 0,Y 340.409,Z 400.894,A -85,B 0,C 180,E1 -14305.261,E2 -14305.261} C_VEL
LIN {X 0,Y 339.829,Z 405.211,A -85,B 0,C 180,E1 -14309.998,E2 -14309.998} C_VEL
LIN {X 0,Y 339.881,Z 407.207,A -85,B 0,C 180,E1 -14311.96,E2 -14311.96} C_VEL
LIN {X 0,Y 343.555,Z 419.655,A -85,B 0,C 180,E1 -14312.71,E2 -14312.71} C_VEL
LIN {X 0,Y 346.417,Z 431.56,A -85,B 0,C 180,E1 -14313.601,E2 -14313.601} C_VEL
LIN {X 0,Y 347.312,Z 436.55,A -85,B 0,C 180,E1 -14314.025,E2 -14314.025} C_VEL
LIN {X 0,Y 346.443,Z 448.331,A -85,B 0,C 180,E1 -14315.032,E2 -14315.032} C_VEL
LIN {X 0,Y 345.263,Z 459.699,A -85,B 0,C 180,E1 -14316.279,E2 -14316.279} C_VEL
LIN {X 0,Y 344.121,Z 469.544,A -85,B 0,C 180,E1 -14317.626,E2 -14317.626} C_VEL
LIN {X 0,Y 343.008,Z 478.506,A -85,B 0,C 180,E1 -14319.134,E2 -14319.134} C_VEL
LIN {X 0,Y 342.088,Z 485.871,A -85,B 0,C 180,E1 -14320.653,E2 -14320.653} C_VEL
LIN {X 0,Y 341.192,Z 493.051,A -85,B 0,C 180,E1 -14322.488,E2 -14322.488} C_VEL
LIN {X 0,Y 340.46,Z 498.788,A -85,B 0,C 180,E1 -14324.34,E2 -14324.34} C_VEL
LIN {X 0,Y 339.966,Z 503.259,A -85,B 0,C 180,E1 -14326.203,E2 -14326.203} C_VEL
LIN {X 0,Y 339.533,Z 506.61,A -85,B 0,C 180,E1 -14328.086,E2 -14328.086} C_VEL
LIN {X 0,Y 339.323,Z 508.27,A -85,B 0,C 180,E1 -14329.35,E2 -14329.35} C_VEL
LIN {X 0,Y 339.169,Z 509.806,A -85,B 0,C 180,E1 -14331.179,E2 -14331.179} C_VEL
LIN {X 0,Y 339.104,Z 510.42,A -85,B 0,C 180,E1 -14333.187,E2 -14333.187} C_VEL
LIN {X 0,Y 339.157,Z 510.193,A -85,B 0,C 180,E1 -14334.481,E2 -14334.481} C_VEL
LIN {X 0,Y 339.242,Z 509.521,A -85,B 0,C 180,E1 -14335.785,E2 -14335.785} C_VEL
LIN {X 0,Y 339.453,Z 508.369,A -85,B 0,C 180,E1 -14337.093,E2 -14337.093} C_VEL
LIN {X 0,Y 339.875,Z 505.645,A -85,B 0,C 180,E1 -14339.071,E2 -14339.071} C_VEL
LIN {X 0,Y 340.388,Z 501.647,A -85,B 0,C 180,E1 -14341.073,E2 -14341.073} C_VEL
LIN {X 0,Y 341.14,Z 496.223,A -85,B 0,C 180,E1 -14343.085,E2 -14343.085} C_VEL
LIN {X 0,Y 342.144,Z 489.092,A -85,B 0,C 180,E1 -14345.107,E2 -14345.107} C_VEL
LIN {X 0,Y 343.167,Z 481.781,A -85,B 0,C 180,E1 -14346.748,E2 -14346.748} C_VEL
LIN {X 0,Y 344.279,Z 473.192,A -85,B 0,C 180,E1 -14348.317,E2 -14348.317} C_VEL
LIN {X 0,Y 345.539,Z 463.349,A -85,B 0,C 180,E1 -14349.771,E2 -14349.771} C_VEL
LIN {X 0,Y 346.695,Z 453.275,A -85,B 0,C 180,E1 -14350.962,E2 -14350.962} C_VEL
LIN {X 0,Y 347.79,Z 441.766,A -85,B 0,C 180,E1 -14352.046,E2 -14352.046} C_VEL
LIN {X 0,Y 347.906,Z 437.327,A -85,B 0,C 180,E1 -14352.413,E2 -14352.413} C_VEL
LIN {X 0,Y 345.144,Z 425.284,A -85,B 0,C 180,E1 -14353.44,E2 -14353.44} C_VEL
LIN {X 0,Y 341.405,Z 412.928,A -85,B 0,C 180,E1 -14354.32,E2 -14354.32} C_VEL
LIN {X 0,Y 339.984,Z 408.248,A -85,B 0,C 180,E1 -14354.611,E2 -14354.611} C_VEL
LIN {X 0,Y 340.06,Z 404.872,A -85,B 0,C 180,E1 -14358.598,E2 -14358.598} C_VEL
LIN {X 0,Y 340.059,Z 404.553,A -85,B 0,C 180,E1 -14358.976,E2 -14358.976} C_VEL
LIN {X 0,Y 339.429,Z 403.82,A -85,B 0,C 180,E1 -14359.958,E2 -14359.958} C_VEL
LIN {X 0,Y 336.673,Z 402.891,A -85,B 0,C 180,E1 -14361.564,E2 -14361.564} C_VEL
LIN {X 0,Y 334.335,Z 402.193,A -85,B 0,C 180,E1 -14362.866,E2 -14362.866} C_VEL
LIN {X 0,Y 333.34,Z 401.534,A -85,B 0,C 180,E1 -14363.869,E2 -14363.869} C_VEL
LIN {X 0,Y 333.264,Z 401.278,A -85,B 0,C 180,E1 -14364.208,E2 -14364.208} C_VEL
LIN {X 0,Y 333.441,Z 398.958,A -85,B 0,C 180,E1 -14367.461,E2 -14367.461} C_VEL
LIN {X 0,Y 333.631,Z 398.931,A -85,B 0,C 180,E1 -14369.725,E2 -14369.725} C_VEL
LIN {X 0,Y 333.722,Z 398.918,A -85,B 0,C 180,E1 -14372.399,E2 -14372.399} C_VEL
LIN {X 0,Y 333.743,Z 398.917,A -85,B 0,C 180,E1 -14375.092,E2 -14375.092} C_VEL
LIN {X 0,Y 333.707,Z 398.92,A -85,B 0,C 180,E1 -14379.021,E2 -14379.021} C_VEL
LIN {X 0,Y 333.777,Z 398.908,A -85,B 0,C 180,E1 -14381.589,E2 -14381.589} C_VEL
LIN {X 0,Y 333.789,Z 398.908,A -85,B 0,C 180,E1 -14385.576,E2 -14385.576} C_VEL
LIN {X 0,Y 333.818,Z 398.903,A -85,B 0,C 180,E1 -14389.078,E2 -14389.078} C_VEL
LIN {X 0,Y 334.008,Z 398.876,A -85,B 0,C 180,E1 -14392.747,E2 -14392.747} C_VEL
LIN {X 0,Y 333.799,Z 398.907,A -85,B 0,C 180,E1 -14395.169,E2 -14395.169} C_VEL
LIN {X 0,Y 334.089,Z 398.87,A -85,B 0,C 180,E1 -14397.589,E2 -14397.589} C_VEL
LIN {X 0,Y 334.248,Z 398.85,A -85,B 0,C 180,E1 -14400,E2 -14400} C_VEL
LIN {X 0,Y 334.121,Z 398.866,A -85,B 0,C 180,E1 -14402.411,E2 -14402.411} C_VEL
LIN {X 0,Y 334.006,Z 398.881,A -85,B 0,C 180,E1 -14407.253,E2 -14407.253} C_VEL
LIN {X 0,Y 333.818,Z 398.902,A -85,B 0,C 180,E1 -14410.923,E2 -14410.923} C_VEL
LIN {X 0,Y 333.79,Z 398.908,A -85,B 0,C 180,E1 -14414.635,E2 -14414.635} C_VEL
LIN {X 0,Y 333.78,Z 398.909,A -85,B 0,C 180,E1 -14418.657,E2 -14418.657} C_VEL
LIN {X 0,Y 333.731,Z 398.918,A -85,B 0,C 180,E1 -14422.276,E2 -14422.276} C_VEL
LIN {X 0,Y 333.72,Z 398.92,A -85,B 0,C 180,E1 -14426.248,E2 -14426.248} C_VEL
LIN {X 0,Y 333.674,Z 398.926,A -85,B 0,C 180,E1 -14428.976,E2 -14428.976} C_VEL
LIN {X 0,Y 333.628,Z 398.929,A -85,B 0,C 180,E1 -14432.589,E2 -14432.589} C_VEL
LIN {X 0,Y 333.662,Z 398.925,A -85,B 0,C 180,E1 -14436.141,E2 -14436.141} C_VEL
LIN {X 0,Y 333.671,Z 398.926,A -85,B 0,C 180,E1 -14439.189,E2 -14439.189} C_VEL
LIN {X 0,Y 333.685,Z 399.064,A -85,B 0,C 180,E1 -14441.162,E2 -14441.162} C_VEL
LIN {X 0,Y 334.481,Z 403.047,A -85,B 0,C 180,E1 -14444.411,E2 -14444.411} C_VEL
LIN {X 0,Y 335.258,Z 407.71,A -85,B 0,C 180,E1 -14447.874,E2 -14447.874} C_VEL
LIN {X 0,Y 336.096,Z 412.482,A -85,B 0,C 180,E1 -14451.151,E2 -14451.151} C_VEL
LIN {X 0,Y 336.434,Z 416.126,A -85,B 0,C 180,E1 -14453.466,E2 -14453.466} C_VEL
LIN {X 0,Y 335.823,Z 420.988,A -85,B 0,C 180,E1 -14456.313,E2 -14456.313} C_VEL
LIN {X 0,Y 334.806,Z 428.388,A -85,B 0,C 180,E1 -14460.446,E2 -14460.446} C_VEL
LIN {X 0,Y 333.974,Z 435.762,A -85,B 0,C 180,E1 -14464.383,E2 -14464.383} C_VEL
LIN {X 0,Y 333.342,Z 442.693,A -85,B 0,C 180,E1 -14467.93,E2 -14467.93} C_VEL
LIN {X 0,Y 336.143,Z 456.297,A -85,B 0,C 180,E1 -14468.652,E2 -14468.652} C_VEL
LIN {X 0,Y 337.755,Z 468.133,A -85,B 0,C 180,E1 -14469.45,E2 -14469.45} C_VEL
LIN {X 0,Y 338.769,Z 480.031,A -85,B 0,C 180,E1 -14470.44,E2 -14470.44} C_VEL
LIN {X 0,Y 339.176,Z 486.888,A -85,B 0,C 180,E1 -14471.112,E2 -14471.112} C_VEL
LIN {X 0,Y 337.804,Z 497.909,A -85,B 0,C 180,E1 -14472.288,E2 -14472.288} C_VEL
LIN {X 0,Y 336.451,Z 508.265,A -85,B 0,C 180,E1 -14473.686,E2 -14473.686} C_VEL
LIN {X 0,Y 335.421,Z 517.006,A -85,B 0,C 180,E1 -14475.138,E2 -14475.138} C_VEL
LIN {X 0,Y 334.229,Z 525.861,A -85,B 0,C 180,E1 -14476.938,E2 -14476.938} C_VEL
LIN {X 0,Y 333.319,Z 533.007,A -85,B 0,C 180,E1 -14478.756,E2 -14478.756} C_VEL
LIN {X 0,Y 332.641,Z 539.562,A -85,B 0,C 180,E1 -14480.885,E2 -14480.885} C_VEL
LIN {X 0,Y 332.289,Z 543.904,A -85,B 0,C 180,E1 -14482.712,E2 -14482.712} C_VEL
LIN {X 0,Y 332.18,Z 546.217,A -85,B 0,C 180,E1 -14483.93,E2 -14483.93} C_VEL
LIN {X 0,Y 332.115,Z 548.067,A -85,B 0,C 180,E1 -14485.147,E2 -14485.147} C_VEL
LIN {X 0,Y 332.057,Z 549.466,A -85,B 0,C 180,E1 -14486.362,E2 -14486.362} C_VEL
LIN {X 0,Y 332.133,Z 551.082,A -85,B 0,C 180,E1 -14488.79,E2 -14488.79} C_VEL
LIN {X 0,Y 332.213,Z 551.271,A -85,B 0,C 180,E1 -14490.002,E2 -14490.002} C_VEL
LIN {X 0,Y 332.167,Z 551.031,A -85,B 0,C 180,E1 -14491.215,E2 -14491.215} C_VEL
LIN {X 0,Y 332.058,Z 549.369,A -85,B 0,C 180,E1 -14493.643,E2 -14493.643} C_VEL
LIN {X 0,Y 332.116,Z 547.91,A -85,B 0,C 180,E1 -14494.858,E2 -14494.858} C_VEL
LIN {X 0,Y 332.221,Z 544.897,A -85,B 0,C 180,E1 -14496.684,E2 -14496.684} C_VEL
LIN {X 0,Y 332.495,Z 540.822,A -85,B 0,C 180,E1 -14498.511,E2 -14498.511} C_VEL
LIN {X 0,Y 333.125,Z 534.56,A -85,B 0,C 180,E1 -14500.64,E2 -14500.64} C_VEL
LIN {X 0,Y 333.885,Z 527.744,A -85,B 0,C 180,E1 -14502.462,E2 -14502.462} C_VEL
LIN {X 0,Y 334.955,Z 519.281,A -85,B 0,C 180,E1 -14504.275,E2 -14504.275} C_VEL
LIN {X 0,Y 335.998,Z 510.381,A -85,B 0,C 180,E1 -14505.809,E2 -14505.809} C_VEL
LIN {X 0,Y 337.271,Z 499.846,A -85,B 0,C 180,E1 -14507.276,E2 -14507.276} C_VEL
LIN {X 0,Y 338.588,Z 489.223,A -85,B 0,C 180,E1 -14508.456,E2 -14508.456} C_VEL
LIN {X 0,Y 338.892,Z 484.498,A -85,B 0,C 180,E1 -14508.909,E2 -14508.909} C_VEL
LIN {X 0,Y 337.808,Z 472.603,A -85,B 0,C 180,E1 -14509.957,E2 -14509.957} C_VEL
LIN {X 0,Y 336.13,Z 459.181,A -85,B 0,C 180,E1 -14510.883,E2 -14510.883} C_VEL
LIN {X 0,Y 333.781,Z 445.854,A -85,B 0,C 180,E1 -14511.581,E2 -14511.581} C_VEL
LIN {X 0,Y 333.334,Z 443.473,A -85,B 0,C 180,E1 -14511.687,E2 -14511.687} C_VEL
LIN {X 0,Y 334.002,Z 435.832,A -85,B 0,C 180,E1 -14515.624,E2 -14515.624} C_VEL
LIN {X 0,Y 334.797,Z 428.371,A -85,B 0,C 180,E1 -14519.56,E2 -14519.56} C_VEL
LIN {X 0,Y 335.811,Z 420.83,A -85,B 0,C 180,E1 -14523.693,E2 -14523.693} C_VEL
LIN {X 0,Y 336.34,Z 417.049,A -85,B 0,C 180,E1 -14525.81,E2 -14525.81} C_VEL
LIN {X 0,Y 336.367,Z 414.298,A -85,B 0,C 180,E1 -14527.442,E2 -14527.442} C_VEL
LIN {X 0,Y 335.4,Z 408.592,A -85,B 0,C 180,E1 -14531.031,E2 -14531.031} C_VEL
LIN {X 0,Y 334.539,Z 403.563,A -85,B 0,C 180,E1 -14534.416,E2 -14534.416} C_VEL
LIN {X 0,Y 333.686,Z 398.922,A -85,B 0,C 180,E1 -14537.829,E2 -14537.829} C_VEL
LIN {X 0,Y 333.659,Z 398.925,A -85,B 0,C 180,E1 -14541.203,E2 -14541.203} C_VEL
LIN {X 0,Y 333.683,Z 398.917,A -85,B 0,C 180,E1 -14543.862,E2 -14543.862} C_VEL
LIN {X 0,Y 333.65,Z 398.922,A -85,B 0,C 180,E1 -14547.414,E2 -14547.414} C_VEL
LIN {X 0,Y 333.697,Z 398.918,A -85,B 0,C 180,E1 -14551.026,E2 -14551.026} C_VEL
LIN {X 0,Y 333.742,Z 398.91,A -85,B 0,C 180,E1 -14553.754,E2 -14553.754} C_VEL
LIN {X 0,Y 333.727,Z 398.912,A -85,B 0,C 180,E1 -14557.914,E2 -14557.914} C_VEL
LIN {X 0,Y 333.801,Z 398.903,A -85,B 0,C 180,E1 -14561.59,E2 -14561.59} C_VEL
LIN {X 0,Y 333.816,Z 398.901,A -85,B 0,C 180,E1 -14565.577,E2 -14565.577} C_VEL
LIN {X 0,Y 333.84,Z 398.898,A -85,B 0,C 180,E1 -14569.078,E2 -14569.078} C_VEL
LIN {X 0,Y 334.012,Z 398.877,A -85,B 0,C 180,E1 -14572.747,E2 -14572.747} C_VEL
LIN {X 0,Y 333.812,Z 398.901,A -85,B 0,C 180,E1 -14575.169,E2 -14575.169} C_VEL
LIN {X 0,Y 334.11,Z 398.865,A -85,B 0,C 180,E1 -14577.589,E2 -14577.589} C_VEL
LIN {X 0,Y 334.233,Z 398.853,A -85,B 0,C 180,E1 -14580,E2 -14580} C_VEL
LIN {X 0,Y 334.11,Z 398.866,A -85,B 0,C 180,E1 -14582.411,E2 -14582.411} C_VEL
LIN {X 0,Y 334.031,Z 398.872,A -85,B 0,C 180,E1 -14587.252,E2 -14587.252} C_VEL
LIN {X 0,Y 333.84,Z 398.897,A -85,B 0,C 180,E1 -14590.922,E2 -14590.922} C_VEL
LIN {X 0,Y 333.815,Z 398.9,A -85,B 0,C 180,E1 -14594.634,E2 -14594.634} C_VEL
LIN {X 0,Y 333.803,Z 398.901,A -85,B 0,C 180,E1 -14598.654,E2 -14598.654} C_VEL
LIN {X 0,Y 333.699,Z 398.915,A -85,B 0,C 180,E1 -14602.278,E2 -14602.278} C_VEL
LIN {X 0,Y 333.741,Z 398.91,A -85,B 0,C 180,E1 -14606.246,E2 -14606.246} C_VEL
LIN {X 0,Y 333.696,Z 398.916,A -85,B 0,C 180,E1 -14608.973,E2 -14608.973} C_VEL
LIN {X 0,Y 333.65,Z 398.919,A -85,B 0,C 180,E1 -14612.586,E2 -14612.586} C_VEL
LIN {X 0,Y 333.682,Z 398.917,A -85,B 0,C 180,E1 -14616.138,E2 -14616.138} C_VEL
LIN {X 0,Y 333.653,Z 398.925,A -85,B 0,C 180,E1 -14619.191,E2 -14619.191} C_VEL
LIN {X 0,Y 333.638,Z 398.922,A -85,B 0,C 180,E1 -14622.499,E2 -14622.499} C_VEL
LIN {X 0,Y 333.628,Z 398.924,A -85,B 0,C 180,E1 -14625.958,E2 -14625.958} C_VEL
LIN {X 0,Y 333.653,Z 398.924,A -85,B 0,C 180,E1 -14629.314,E2 -14629.314} C_VEL
LIN {X 0,Y 333.671,Z 398.923,A -85,B 0,C 180,E1 -14633.167,E2 -14633.167} C_VEL
LIN {X 0,Y 333.68,Z 398.92,A -85,B 0,C 180,E1 -14635.34,E2 -14635.34} C_VEL
LIN {X 0,Y 333.696,Z 398.915,A -85,B 0,C 180,E1 -14639.636,E2 -14639.636} C_VEL
LIN {X 0,Y 333.745,Z 398.911,A -85,B 0,C 180,E1 -14642.399,E2 -14642.399} C_VEL
LIN {X 0,Y 333.732,Z 398.914,A -85,B 0,C 180,E1 -14645.089,E2 -14645.089} C_VEL
LIN {X 0,Y 333.69,Z 398.919,A -85,B 0,C 180,E1 -14649.018,E2 -14649.018} C_VEL
LIN {X 0,Y 333.798,Z 398.902,A -85,B 0,C 180,E1 -14651.588,E2 -14651.588} C_VEL
LIN {X 0,Y 333.812,Z 398.901,A -85,B 0,C 180,E1 -14655.575,E2 -14655.575} C_VEL
LIN {X 0,Y 333.603,Z 398.928,A -85,B 0,C 180,E1 -14659.068,E2 -14659.068} C_VEL
LIN {X 0,Y 333.397,Z 398.955,A -85,B 0,C 180,E1 -14661.512,E2 -14661.512} C_VEL
LIN {X 0,Y 333.3,Z 399.664,A -85,B 0,C 180,E1 -14662.729,E2 -14662.729} C_VEL
LIN {X 0,Y 333.378,Z 401.7,A -85,B 0,C 180,E1 -14665.161,E2 -14665.161} C_VEL
LIN {X 0,Y 332.774,Z 405.987,A -85,B 0,C 180,E1 -14669.998,E2 -14669.998} C_VEL
LIN {X 0,Y 332.754,Z 407.459,A -85,B 0,C 180,E1 -14671.51,E2 -14671.51} C_VEL
LIN {X 0,Y 336.818,Z 420.88,A -85,B 0,C 180,E1 -14672.352,E2 -14672.352} C_VEL
LIN {X 0,Y 339.713,Z 433.205,A -85,B 0,C 180,E1 -14673.311,E2 -14673.311} C_VEL
LIN {X 0,Y 340.473,Z 437.209,A -85,B 0,C 180,E1 -14673.671,E2 -14673.671} C_VEL
LIN {X 0,Y 339.753,Z 447.556,A -85,B 0,C 180,E1 -14674.57,E2 -14674.57} C_VEL
LIN {X 0,Y 338.64,Z 458.675,A -85,B 0,C 180,E1 -14675.773,E2 -14675.773} C_VEL
LIN {X 0,Y 337.356,Z 468.995,A -85,B 0,C 180,E1 -14677.178,E2 -14677.178} C_VEL
LIN {X 0,Y 336.227,Z 478.099,A -85,B 0,C 180,E1 -14678.714,E2 -14678.714} C_VEL
LIN {X 0,Y 335.184,Z 485.993,A -85,B 0,C 180,E1 -14680.347,E2 -14680.347} C_VEL
LIN {X 0,Y 334.272,Z 492.965,A -85,B 0,C 180,E1 -14682.134,E2 -14682.134} C_VEL
LIN {X 0,Y 333.434,Z 499.197,A -85,B 0,C 180,E1 -14684.171,E2 -14684.171} C_VEL
LIN {X 0,Y 332.961,Z 503.366,A -85,B 0,C 180,E1 -14685.923,E2 -14685.923} C_VEL
LIN {X 0,Y 332.491,Z 507,A -85,B 0,C 180,E1 -14687.976,E2 -14687.976} C_VEL
LIN {X 0,Y 332.173,Z 509.174,A -85,B 0,C 180,E1 -14689.784,E2 -14689.784} C_VEL
LIN {X 0,Y 332.085,Z 510.352,A -85,B 0,C 180,E1 -14691.38,E2 -14691.38} C_VEL
LIN {X 0,Y 332.038,Z 510.806,A -85,B 0,C 180,E1 -14693.71,E2 -14693.71} C_VEL
LIN {X 0,Y 332.108,Z 510.445,A -85,B 0,C 180,E1 -14695.036,E2 -14695.036} C_VEL
LIN {X 0,Y 332.416,Z 508.597,A -85,B 0,C 180,E1 -14697.38,E2 -14697.38} C_VEL
LIN {X 0,Y 332.79,Z 506.362,A -85,B 0,C 180,E1 -14699.057,E2 -14699.057} C_VEL
LIN {X 0,Y 333.319,Z 502.463,A -85,B 0,C 180,E1 -14701.1,E2 -14701.1} C_VEL
LIN {X 0,Y 334.098,Z 497.148,A -85,B 0,C 180,E1 -14703.153,E2 -14703.153} C_VEL
LIN {X 0,Y 335.125,Z 490.525,A -85,B 0,C 180,E1 -14705.127,E2 -14705.127} C_VEL
LIN {X 0,Y 336.23,Z 482.818,A -85,B 0,C 180,E1 -14706.934,E2 -14706.934} C_VEL
LIN {X 0,Y 337.49,Z 473.625,A -85,B 0,C 180,E1 -14708.658,E2 -14708.658} C_VEL
LIN {X 0,Y 338.7,Z 464.573,A -85,B 0,C 180,E1 -14710.03,E2 -14710.03} C_VEL
LIN {X 0,Y 339.871,Z 454.875,A -85,B 0,C 180,E1 -14711.229,E2 -14711.229} C_VEL
LIN {X 0,Y 341.05,Z 443.527,A -85,B 0,C 180,E1 -14712.343,E2 -14712.343} C_VEL
LIN {X 0,Y 341.27,Z 439.014,A -85,B 0,C 180,E1 -14712.73,E2 -14712.73} C_VEL
LIN {X 0,Y 338.536,Z 426.92,A -85,B 0,C 180,E1 -14713.808,E2 -14713.808} C_VEL
LIN {X 0,Y 334.968,Z 415.041,A -85,B 0,C 180,E1 -14714.705,E2 -14714.705} C_VEL
LIN {X 0,Y 332.925,Z 408.711,A -85,B 0,C 180,E1 -14715.128,E2 -14715.128} C_VEL
LIN {X 0,Y 333.048,Z 405.359,A -85,B 0,C 180,E1 -14719.144,E2 -14719.144} C_VEL
LIN {X 0,Y 333.203,Z 402.807,A -85,B 0,C 180,E1 -14722.289,E2 -14722.289} C_VEL
LIN {X 0,Y 333.264,Z 401.278,A -85,B 0,C 180,E1 -14724.208,E2 -14724.208} C_VEL
LIN {X 0,Y 332.635,Z 400.622,A -85,B 0,C 180,E1 -14725.211,E2 -14725.211} C_VEL
LIN {X 0,Y 329.906,Z 400.024,A -85,B 0,C 180,E1 -14726.855,E2 -14726.855} C_VEL
LIN {X 0,Y 327.599,Z 399.851,A -85,B 0,C 180,E1 -14728.189,E2 -14728.189} C_VEL
LIN {X 0,Y 326.627,Z 399.815,A -85,B 0,C 180,E1 -14729.22,E2 -14729.22} C_VEL
LIN {X 0,Y 326.557,Z 399.811,A -85,B 0,C 180,E1 -14729.568,E2 -14729.568} C_VEL
LIN {X 0,Y 326.666,Z 399.796,A -85,B 0,C 180,E1 -14733.141,E2 -14733.141} C_VEL
LIN {X 0,Y 326.68,Z 399.796,A -85,B 0,C 180,E1 -14737.217,E2 -14737.217} C_VEL
LIN {X 0,Y 326.726,Z 399.787,A -85,B 0,C 180,E1 -14741.176,E2 -14741.176} C_VEL
LIN {X 0,Y 326.744,Z 399.785,A -85,B 0,C 180,E1 -14745.432,E2 -14745.432} C_VEL
LIN {X 0,Y 326.754,Z 399.784,A -85,B 0,C 180,E1 -14748.838,E2 -14748.838} C_VEL
LIN {X 0,Y 326.962,Z 399.755,A -85,B 0,C 180,E1 -14752.59,E2 -14752.59} C_VEL
LIN {X 0,Y 326.765,Z 399.784,A -85,B 0,C 180,E1 -14755.065,E2 -14755.065} C_VEL
LIN {X 0,Y 327.03,Z 399.749,A -85,B 0,C 180,E1 -14757.537,E2 -14757.537} C_VEL
LIN {X 0,Y 327.199,Z 399.728,A -85,B 0,C 180,E1 -14760,E2 -14760} C_VEL
LIN {X 0,Y 327.058,Z 399.746,A -85,B 0,C 180,E1 -14762.463,E2 -14762.463} C_VEL
LIN {X 0,Y 326.977,Z 399.757,A -85,B 0,C 180,E1 -14766.17,E2 -14766.17} C_VEL
LIN {X 0,Y 326.896,Z 399.768,A -85,B 0,C 180,E1 -14768.656,E2 -14768.656} C_VEL
LIN {X 0,Y 326.719,Z 399.788,A -85,B 0,C 180,E1 -14772.422,E2 -14772.422} C_VEL
LIN {X 0,Y 326.736,Z 399.787,A -85,B 0,C 180,E1 -14774.959,E2 -14774.959} C_VEL
LIN {X 0,Y 326.746,Z 399.785,A -85,B 0,C 180,E1 -14778.855,E2 -14778.855} C_VEL
LIN {X 0,Y 326.68,Z 399.796,A -85,B 0,C 180,E1 -14782.783,E2 -14782.783} C_VEL
LIN {X 0,Y 326.667,Z 399.799,A -85,B 0,C 180,E1 -14786.859,E2 -14786.859} C_VEL
LIN {X 0,Y 326.618,Z 399.806,A -85,B 0,C 180,E1 -14790.611,E2 -14790.611} C_VEL
LIN {X 0,Y 326.592,Z 399.806,A -85,B 0,C 180,E1 -14794.021,E2 -14794.021} C_VEL
LIN {X 0,Y 326.615,Z 399.803,A -85,B 0,C 180,E1 -14797.241,E2 -14797.241} C_VEL
LIN {X 0,Y 326.626,Z 399.822,A -85,B 0,C 180,E1 -14800.452,E2 -14800.452} C_VEL
LIN {X 0,Y 327.27,Z 403.278,A -85,B 0,C 180,E1 -14803.408,E2 -14803.408} C_VEL
LIN {X 0,Y 328.037,Z 407.562,A -85,B 0,C 180,E1 -14806.755,E2 -14806.755} C_VEL
LIN {X 0,Y 328.9,Z 412.487,A -85,B 0,C 180,E1 -14810.287,E2 -14810.287} C_VEL
LIN {X 0,Y 329.354,Z 415.258,A -85,B 0,C 180,E1 -14812.142,E2 -14812.142} C_VEL
LIN {X 0,Y 329.322,Z 418.522,A -85,B 0,C 180,E1 -14814.189,E2 -14814.189} C_VEL
LIN {X 0,Y 328.4,Z 424.392,A -85,B 0,C 180,E1 -14817.658,E2 -14817.658} C_VEL
LIN {X 0,Y 327.594,Z 430.489,A -85,B 0,C 180,E1 -14821.107,E2 -14821.107} C_VEL
LIN {X 0,Y 326.868,Z 436.839,A -85,B 0,C 180,E1 -14824.562,E2 -14824.562} C_VEL
LIN {X 0,Y 326.34,Z 442.093,A -85,B 0,C 180,E1 -14827.359,E2 -14827.359} C_VEL
LIN {X 0,Y 329.511,Z 457.546,A -85,B 0,C 180,E1 -14828.262,E2 -14828.262} C_VEL
LIN {X 0,Y 331.179,Z 470.535,A -85,B 0,C 180,E1 -14829.2,E2 -14829.2} C_VEL
LIN {X 0,Y 332.054,Z 481.874,A -85,B 0,C 180,E1 -14830.209,E2 -14830.209} C_VEL
LIN {X 0,Y 332.268,Z 488.246,A -85,B 0,C 180,E1 -14830.865,E2 -14830.865} C_VEL
LIN {X 0,Y 330.698,Z 500.03,A -85,B 0,C 180,E1 -14832.215,E2 -14832.215} C_VEL
LIN {X 0,Y 329.395,Z 509.56,A -85,B 0,C 180,E1 -14833.581,E2 -14833.581} C_VEL
LIN {X 0,Y 328.293,Z 518.295,A -85,B 0,C 180,E1 -14835.117,E2 -14835.117} C_VEL
LIN {X 0,Y 327.094,Z 526.797,A -85,B 0,C 180,E1 -14836.964,E2 -14836.964} C_VEL
LIN {X 0,Y 326.187,Z 533.661,A -85,B 0,C 180,E1 -14838.821,E2 -14838.821} C_VEL
LIN {X 0,Y 325.605,Z 539.175,A -85,B 0,C 180,E1 -14840.686,E2 -14840.686} C_VEL
LIN {X 0,Y 325.215,Z 543.506,A -85,B 0,C 180,E1 -14842.553,E2 -14842.553} C_VEL
LIN {X 0,Y 325.102,Z 546.068,A -85,B 0,C 180,E1 -14843.947,E2 -14843.947} C_VEL
LIN {X 0,Y 324.986,Z 549.051,A -85,B 0,C 180,E1 -14846.283,E2 -14846.283} C_VEL
LIN {X 0,Y 325.04,Z 550.657,A -85,B 0,C 180,E1 -14848.763,E2 -14848.763} C_VEL
LIN {X 0,Y 325.138,Z 550.838,A -85,B 0,C 180,E1 -14850.002,E2 -14850.002} C_VEL
LIN {X 0,Y 325.073,Z 550.591,A -85,B 0,C 180,E1 -14851.241,E2 -14851.241} C_VEL
LIN {X 0,Y 324.987,Z 548.921,A -85,B 0,C 180,E1 -14853.722,E2 -14853.722} C_VEL
LIN {X 0,Y 325.085,Z 545.843,A -85,B 0,C 180,E1 -14856.025,E2 -14856.025} C_VEL
LIN {X 0,Y 325.304,Z 541.799,A -85,B 0,C 180,E1 -14858.075,E2 -14858.075} C_VEL
LIN {X 0,Y 325.805,Z 536.951,A -85,B 0,C 180,E1 -14859.939,E2 -14859.939} C_VEL
LIN {X 0,Y 326.435,Z 530.827,A -85,B 0,C 180,E1 -14861.804,E2 -14861.804} C_VEL
LIN {X 0,Y 327.493,Z 523.228,A -85,B 0,C 180,E1 -14863.656,E2 -14863.656} C_VEL
LIN {X 0,Y 328.656,Z 514.365,A -85,B 0,C 180,E1 -14865.387,E2 -14865.387} C_VEL
LIN {X 0,Y 329.715,Z 504.91,A -85,B 0,C 180,E1 -14866.885,E2 -14866.885} C_VEL
LIN {X 0,Y 331.116,Z 494.207,A -85,B 0,C 180,E1 -14868.247,E2 -14868.247} C_VEL
LIN {X 0,Y 332.005,Z 485.43,A -85,B 0,C 180,E1 -14869.156,E2 -14869.156} C_VEL
LIN {X 0,Y 330.93,Z 473.159,A -85,B 0,C 180,E1 -14870.29,E2 -14870.29} C_VEL
LIN {X 0,Y 329.399,Z 460.469,A -85,B 0,C 180,E1 -14871.207,E2 -14871.207} C_VEL
LIN {X 0,Y 327.006,Z 446.848,A -85,B 0,C 180,E1 -14871.969,E2 -14871.969} C_VEL
LIN {X 0,Y 326.314,Z 443.029,A -85,B 0,C 180,E1 -14872.163,E2 -14872.163} C_VEL
LIN {X 0,Y 327.038,Z 435.527,A -85,B 0,C 180,E1 -14876.141,E2 -14876.141} C_VEL
LIN {X 0,Y 327.911,Z 427.98,A -85,B 0,C 180,E1 -14880.245,E2 -14880.245} C_VEL
LIN {X 0,Y 328.785,Z 421.69,A -85,B 0,C 180,E1 -14883.766,E2 -14883.766} C_VEL
LIN {X 0,Y 329.396,Z 416.684,A -85,B 0,C 180,E1 -14886.687,E2 -14886.687} C_VEL
LIN {X 0,Y 328.978,Z 413.034,A -85,B 0,C 180,E1 -14888.966,E2 -14888.966} C_VEL
LIN {X 0,Y 328.111,Z 407.834,A -85,B 0,C 180,E1 -14892.387,E2 -14892.387} C_VEL
LIN {X 0,Y 327.388,Z 403.956,A -85,B 0,C 180,E1 -14895.108,E2 -14895.108} C_VEL
LIN {X 0,Y 326.656,Z 399.796,A -85,B 0,C 180,E1 -14898.268,E2 -14898.268} C_VEL
LIN {X 0,Y 326.63,Z 399.8,A -85,B 0,C 180,E1 -14901.392,E2 -14901.392} C_VEL
LIN {X 0,Y 326.627,Z 399.802,A -85,B 0,C 180,E1 -14904.852,E2 -14904.852} C_VEL
LIN {X 0,Y 326.615,Z 399.798,A -85,B 0,C 180,E1 -14907.456,E2 -14907.456} C_VEL
LIN {X 0,Y 326.655,Z 399.796,A -85,B 0,C 180,E1 -14910.34,E2 -14910.34} C_VEL
LIN {X 0,Y 326.697,Z 399.792,A -85,B 0,C 180,E1 -14914.517,E2 -14914.517} C_VEL
LIN {X 0,Y 326.653,Z 399.799,A -85,B 0,C 180,E1 -14918.546,E2 -14918.546} C_VEL
LIN {X 0,Y 326.752,Z 399.781,A -85,B 0,C 180,E1 -14921.178,E2 -14921.178} C_VEL
LIN {X 0,Y 326.771,Z 399.779,A -85,B 0,C 180,E1 -14925.433,E2 -14925.433} C_VEL
LIN {X 0,Y 326.777,Z 399.779,A -85,B 0,C 180,E1 -14928.839,E2 -14928.839} C_VEL
LIN {X 0,Y 326.965,Z 399.757,A -85,B 0,C 180,E1 -14932.59,E2 -14932.59} C_VEL
LIN {X 0,Y 326.779,Z 399.777,A -85,B 0,C 180,E1 -14935.065,E2 -14935.065} C_VEL
LIN {X 0,Y 327.051,Z 399.744,A -85,B 0,C 180,E1 -14937.537,E2 -14937.537} C_VEL
LIN {X 0,Y 327.185,Z 399.731,A -85,B 0,C 180,E1 -14940,E2 -14940} C_VEL
LIN {X 0,Y 327.051,Z 399.744,A -85,B 0,C 180,E1 -14942.463,E2 -14942.463} C_VEL
LIN {X 0,Y 326.974,Z 399.749,A -85,B 0,C 180,E1 -14946.701,E2 -14946.701} C_VEL
LIN {X 0,Y 326.821,Z 399.776,A -85,B 0,C 180,E1 -14949.906,E2 -14949.906} C_VEL
LIN {X 0,Y 326.766,Z 399.783,A -85,B 0,C 180,E1 -14953.685,E2 -14953.685} C_VEL
LIN {X 0,Y 326.706,Z 399.789,A -85,B 0,C 180,E1 -14957.527,E2 -14957.527} C_VEL
LIN {X 0,Y 326.669,Z 399.789,A -85,B 0,C 180,E1 -14960.134,E2 -14960.134} C_VEL
LIN {X 0,Y 326.659,Z 399.793,A -85,B 0,C 180,E1 -14964.128,E2 -14964.128} C_VEL
LIN {X 0,Y 326.689,Z 399.789,A -85,B 0,C 180,E1 -14966.857,E2 -14966.857} C_VEL
LIN {X 0,Y 326.641,Z 399.793,A -85,B 0,C 180,E1 -14970.609,E2 -14970.609} C_VEL
LIN {X 0,Y 326.613,Z 399.797,A -85,B 0,C 180,E1 -14974.019,E2 -14974.019} C_VEL
LIN {X 0,Y 326.634,Z 399.799,A -85,B 0,C 180,E1 -14977.238,E2 -14977.238} C_VEL
LIN {X 0,Y 326.584,Z 399.805,A -85,B 0,C 180,E1 -14981.13,E2 -14981.13} C_VEL
LIN {X 0,Y 326.561,Z 399.804,A -85,B 0,C 180,E1 -14984.747,E2 -14984.747} C_VEL
LIN {X 0,Y 326.583,Z 399.801,A -85,B 0,C 180,E1 -14988.153,E2 -14988.153} C_VEL
LIN {X 0,Y 326.604,Z 399.8,A -85,B 0,C 180,E1 -14991.387,E2 -14991.387} C_VEL
LIN {X 0,Y 326.625,Z 399.8,A -85,B 0,C 180,E1 -14994.85,E2 -14994.85} C_VEL
LIN {X 0,Y 326.613,Z 399.799,A -85,B 0,C 180,E1 -14997.454,E2 -14997.454} C_VEL
LIN {X 0,Y 326.653,Z 399.793,A -85,B 0,C 180,E1 -15000.338,E2 -15000.338} C_VEL
LIN {X 0,Y 326.695,Z 399.791,A -85,B 0,C 180,E1 -15004.515,E2 -15004.515} C_VEL
LIN {X 0,Y 326.653,Z 399.797,A -85,B 0,C 180,E1 -15008.544,E2 -15008.544} C_VEL
LIN {X 0,Y 326.749,Z 399.782,A -85,B 0,C 180,E1 -15011.176,E2 -15011.176} C_VEL
LIN {X 0,Y 326.767,Z 399.779,A -85,B 0,C 180,E1 -15015.431,E2 -15015.431} C_VEL
LIN {X 0,Y 326.582,Z 399.805,A -85,B 0,C 180,E1 -15018.83,E2 -15018.83} C_VEL
LIN {X 0,Y 326.363,Z 399.832,A -85,B 0,C 180,E1 -15021.328,E2 -15021.328} C_VEL
LIN {X 0,Y 326.283,Z 400.442,A -85,B 0,C 180,E1 -15022.572,E2 -15022.572} C_VEL
LIN {X 0,Y 326.349,Z 402.528,A -85,B 0,C 180,E1 -15025.056,E2 -15025.056} C_VEL
LIN {X 0,Y 325.726,Z 406.869,A -85,B 0,C 180,E1 -15029.998,E2 -15029.998} C_VEL
LIN {X 0,Y 325.707,Z 407.798,A -85,B 0,C 180,E1 -15031.041,E2 -15031.041} C_VEL
LIN {X 0,Y 329.949,Z 421.739,A -85,B 0,C 180,E1 -15031.955,E2 -15031.955} C_VEL
LIN {X 0,Y 332.967,Z 434.636,A -85,B 0,C 180,E1 -15032.999,E2 -15032.999} C_VEL
LIN {X 0,Y 333.718,Z 439.596,A -85,B 0,C 180,E1 -15033.451,E2 -15033.451} C_VEL
LIN {X 0,Y 332.662,Z 451.264,A -85,B 0,C 180,E1 -15034.542,E2 -15034.542} C_VEL
LIN {X 0,Y 331.437,Z 462.441,A -85,B 0,C 180,E1 -15035.866,E2 -15035.866} C_VEL
LIN {X 0,Y 330.165,Z 472.367,A -85,B 0,C 180,E1 -15037.335,E2 -15037.335} C_VEL
LIN {X 0,Y 328.997,Z 480.937,A -85,B 0,C 180,E1 -15038.907,E2 -15038.907} C_VEL
LIN {X 0,Y 327.857,Z 489.177,A -85,B 0,C 180,E1 -15040.777,E2 -15040.777} C_VEL
LIN {X 0,Y 327.072,Z 494.97,A -85,B 0,C 180,E1 -15042.406,E2 -15042.406} C_VEL
LIN {X 0,Y 326.347,Z 500.356,A -85,B 0,C 180,E1 -15044.282,E2 -15044.282} C_VEL
LIN {X 0,Y 325.81,Z 504.783,A -85,B 0,C 180,E1 -15046.283,E2 -15046.283} C_VEL
LIN {X 0,Y 325.381,Z 507.778,A -85,B 0,C 180,E1 -15048.127,E2 -15048.127} C_VEL
LIN {X 0,Y 325.046,Z 510.063,A -85,B 0,C 180,E1 -15050.236,E2 -15050.236} C_VEL
LIN {X 0,Y 324.988,Z 510.873,A -85,B 0,C 180,E1 -15051.582,E2 -15051.582} C_VEL
LIN {X 0,Y 324.929,Z 511.245,A -85,B 0,C 180,E1 -15052.91,E2 -15052.91} C_VEL
LIN {X 0,Y 324.999,Z 511.011,A -85,B 0,C 180,E1 -15054.737,E2 -15054.737} C_VEL
LIN {X 0,Y 325.255,Z 509.562,A -85,B 0,C 180,E1 -15056.982,E2 -15056.982} C_VEL
LIN {X 0,Y 325.704,Z 507.056,A -85,B 0,C 180,E1 -15059.042,E2 -15059.042} C_VEL
LIN {X 0,Y 326.251,Z 503.289,A -85,B 0,C 180,E1 -15061.128,E2 -15061.128} C_VEL
LIN {X 0,Y 327.16,Z 497.501,A -85,B 0,C 180,E1 -15063.427,E2 -15063.427} C_VEL
LIN {X 0,Y 328.184,Z 491.289,A -85,B 0,C 180,E1 -15065.32,E2 -15065.32} C_VEL
LIN {X 0,Y 329.243,Z 484.081,A -85,B 0,C 180,E1 -15067.083,E2 -15067.083} C_VEL
LIN {X 0,Y 330.575,Z 475.076,A -85,B 0,C 180,E1 -15068.838,E2 -15068.838} C_VEL
LIN {X 0,Y 331.9,Z 465.566,A -85,B 0,C 180,E1 -15070.333,E2 -15070.333} C_VEL
LIN {X 0,Y 333.191,Z 455.307,A -85,B 0,C 180,E1 -15071.634,E2 -15071.634} C_VEL
LIN {X 0,Y 334.393,Z 444.242,A -85,B 0,C 180,E1 -15072.744,E2 -15072.744} C_VEL
LIN {X 0,Y 334.551,Z 440.246,A -85,B 0,C 180,E1 -15073.103,E2 -15073.103} C_VEL
LIN {X 0,Y 332.019,Z 428.893,A -85,B 0,C 180,E1 -15074.167,E2 -15074.167} C_VEL
LIN {X 0,Y 328.454,Z 416.734,A -85,B 0,C 180,E1 -15075.133,E2 -15075.133} C_VEL
LIN {X 0,Y 325.903,Z 409.176,A -85,B 0,C 180,E1 -15075.664,E2 -15075.664} C_VEL
LIN {X 0,Y 326.022,Z 405.881,A -85,B 0,C 180,E1 -15079.706,E2 -15079.706} C_VEL
LIN {X 0,Y 326.195,Z 403.336,A -85,B 0,C 180,E1 -15082.896,E2 -15082.896} C_VEL
LIN {X 0,Y 326.332,Z 400.984,A -85,B 0,C 180,E1 -15085.948,E2 -15085.948} C_VEL
LIN {X 0,Y 326.409,Z 399.864,A -85,B 0,C 180,E1 -15087.433,E2 -15087.433} C_VEL
LIN {X 0,Y 326.557,Z 399.811,A -85,B 0,C 180,E1 -15089.568,E2 -15089.568} C_VEL
LIN {X 0,Y 325.919,Z 399.89,A -85,B 0,C 180,E1 -15090.598,E2 -15090.598} C_VEL
LIN {X 0,Y 323.099,Z 400.24,A -85,B 0,C 180,E1 -15092.274,E2 -15092.274} C_VEL
LIN {X 0,Y 320.702,Z 400.54,A -85,B 0,C 180,E1 -15093.631,E2 -15093.631} C_VEL
LIN {X 0,Y 319.682,Z 400.666,A -85,B 0,C 180,E1 -15094.682,E2 -15094.682} C_VEL
LIN {X 0,Y 319.605,Z 400.676,A -85,B 0,C 180,E1 -15095.038,E2 -15095.038} C_VEL
LIN {X 0,Y 319.635,Z 400.671,A -85,B 0,C 180,E1 -15098.051,E2 -15098.051} C_VEL
LIN {X 0,Y 319.688,Z 400.664,A -85,B 0,C 180,E1 -15100.952,E2 -15100.952} C_VEL
LIN {X 0,Y 319.712,Z 400.661,A -85,B 0,C 180,E1 -15105.275,E2 -15105.275} C_VEL
LIN {X 0,Y 319.741,Z 400.654,A -85,B 0,C 180,E1 -15109.872,E2 -15109.872} C_VEL
LIN {X 0,Y 319.915,Z 400.633,A -85,B 0,C 180,E1 -15112.426,E2 -15112.426} C_VEL
LIN {X 0,Y 319.734,Z 400.659,A -85,B 0,C 180,E1 -15114.956,E2 -15114.956} C_VEL
LIN {X 0,Y 319.974,Z 400.628,A -85,B 0,C 180,E1 -15117.482,E2 -15117.482} C_VEL
LIN {X 0,Y 320.15,Z 400.606,A -85,B 0,C 180,E1 -15120,E2 -15120} C_VEL
LIN {X 0,Y 319.999,Z 400.625,A -85,B 0,C 180,E1 -15122.518,E2 -15122.518} C_VEL
LIN {X 0,Y 319.933,Z 400.635,A -85,B 0,C 180,E1 -15126.306,E2 -15126.306} C_VEL
LIN {X 0,Y 319.824,Z 400.648,A -85,B 0,C 180,E1 -15128.849,E2 -15128.849} C_VEL
LIN {X 0,Y 319.666,Z 400.667,A -85,B 0,C 180,E1 -15132.701,E2 -15132.701} C_VEL
LIN {X 0,Y 319.681,Z 400.666,A -85,B 0,C 180,E1 -15135.297,E2 -15135.297} C_VEL
LIN {X 0,Y 319.674,Z 400.667,A -85,B 0,C 180,E1 -15139.255,E2 -15139.255} C_VEL
LIN {X 0,Y 319.628,Z 400.674,A -85,B 0,C 180,E1 -15143.315,E2 -15143.315} C_VEL
LIN {X 0,Y 319.619,Z 400.677,A -85,B 0,C 180,E1 -15146.09,E2 -15146.09} C_VEL
LIN {X 0,Y 319.564,Z 400.684,A -85,B 0,C 180,E1 -15148.936,E2 -15148.936} C_VEL
LIN {X 0,Y 319.515,Z 400.69,A -85,B 0,C 180,E1 -15151.864,E2 -15151.864} C_VEL
LIN {X 0,Y 319.565,Z 400.681,A -85,B 0,C 180,E1 -15155.545,E2 -15155.545} C_VEL
LIN {X 0,Y 319.586,Z 400.678,A -85,B 0,C 180,E1 -15158.006,E2 -15158.006} C_VEL
LIN {X 0,Y 319.576,Z 400.698,A -85,B 0,C 180,E1 -15159.809,E2 -15159.809} C_VEL
LIN {X 0,Y 320.388,Z 405.04,A -85,B 0,C 180,E1 -15163.629,E2 -15163.629} C_VEL
LIN {X 0,Y 321.195,Z 409.688,A -85,B 0,C 180,E1 -15167.293,E2 -15167.293} C_VEL
LIN {X 0,Y 322.043,Z 414.446,A -85,B 0,C 180,E1 -15170.742,E2 -15170.742} C_VEL
LIN {X 0,Y 322.428,Z 418.013,A -85,B 0,C 180,E1 -15173.151,E2 -15173.151} C_VEL
LIN {X 0,Y 321.833,Z 422.75,A -85,B 0,C 180,E1 -15176.081,E2 -15176.081} C_VEL
LIN {X 0,Y 320.693,Z 430.24,A -85,B 0,C 180,E1 -15180.46,E2 -15180.46} C_VEL
LIN {X 0,Y 319.856,Z 437.022,A -85,B 0,C 180,E1 -15184.273,E2 -15184.273} C_VEL
LIN {X 0,Y 319.342,Z 441.897,A -85,B 0,C 180,E1 -15186.828,E2 -15186.828} C_VEL
LIN {X 0,Y 322.282,Z 455.384,A -85,B 0,C 180,E1 -15187.613,E2 -15187.613} C_VEL
LIN {X 0,Y 324.027,Z 467.245,A -85,B 0,C 180,E1 -15188.473,E2 -15188.473} C_VEL
LIN {X 0,Y 325.11,Z 480.071,A -85,B 0,C 180,E1 -15189.612,E2 -15189.612} C_VEL
LIN {X 0,Y 325.546,Z 488.051,A -85,B 0,C 180,E1 -15190.454,E2 -15190.454} C_VEL
LIN {X 0,Y 323.927,Z 499.79,A -85,B 0,C 180,E1 -15191.83,E2 -15191.83} C_VEL
LIN {X 0,Y 322.553,Z 509.286,A -85,B 0,C 180,E1 -15193.223,E2 -15193.223} C_VEL
LIN {X 0,Y 321.422,Z 517.992,A -85,B 0,C 180,E1 -15194.791,E2 -15194.791} C_VEL
LIN {X 0,Y 320.147,Z 526.462,A -85,B 0,C 180,E1 -15196.676,E2 -15196.676} C_VEL
LIN {X 0,Y 319.162,Z 533.306,A -85,B 0,C 180,E1 -15198.572,E2 -15198.572} C_VEL
LIN {X 0,Y 318.568,Z 538.804,A -85,B 0,C 180,E1 -15200.479,E2 -15200.479} C_VEL
LIN {X 0,Y 318.165,Z 543.119,A -85,B 0,C 180,E1 -15202.386,E2 -15202.386} C_VEL
LIN {X 0,Y 318.01,Z 545.927,A -85,B 0,C 180,E1 -15203.99,E2 -15203.99} C_VEL
LIN {X 0,Y 317.915,Z 548.638,A -85,B 0,C 180,E1 -15206.2,E2 -15206.2} C_VEL
LIN {X 0,Y 317.946,Z 550.232,A -85,B 0,C 180,E1 -15208.736,E2 -15208.736} C_VEL
LIN {X 0,Y 318.049,Z 550.403,A -85,B 0,C 180,E1 -15210.002,E2 -15210.002} C_VEL
LIN {X 0,Y 317.979,Z 550.152,A -85,B 0,C 180,E1 -15211.269,E2 -15211.269} C_VEL
LIN {X 0,Y 317.916,Z 548.472,A -85,B 0,C 180,E1 -15213.805,E2 -15213.805} C_VEL
LIN {X 0,Y 318.002,Z 545.648,A -85,B 0,C 180,E1 -15215.998,E2 -15215.998} C_VEL
LIN {X 0,Y 318.244,Z 541.315,A -85,B 0,C 180,E1 -15218.255,E2 -15218.255} C_VEL
LIN {X 0,Y 318.759,Z 536.45,A -85,B 0,C 180,E1 -15220.161,E2 -15220.161} C_VEL
LIN {X 0,Y 319.451,Z 530.307,A -85,B 0,C 180,E1 -15222.066,E2 -15222.066} C_VEL
LIN {X 0,Y 320.542,Z 522.683,A -85,B 0,C 180,E1 -15223.958,E2 -15223.958} C_VEL
LIN {X 0,Y 321.726,Z 514.158,A -85,B 0,C 180,E1 -15225.658,E2 -15225.658} C_VEL
LIN {X 0,Y 322.865,Z 504.285,A -85,B 0,C 180,E1 -15227.255,E2 -15227.255} C_VEL
LIN {X 0,Y 324.341,Z 493.538,A -85,B 0,C 180,E1 -15228.642,E2 -15228.642} C_VEL
LIN {X 0,Y 325.09,Z 486.289,A -85,B 0,C 180,E1 -15229.416,E2 -15229.416} C_VEL
LIN {X 0,Y 324.034,Z 473.555,A -85,B 0,C 180,E1 -15230.641,E2 -15230.641} C_VEL
LIN {X 0,Y 322.55,Z 460.854,A -85,B 0,C 180,E1 -15231.603,E2 -15231.603} C_VEL
LIN {X 0,Y 320.15,Z 447.124,A -85,B 0,C 180,E1 -15232.405,E2 -15232.405} C_VEL
LIN {X 0,Y 319.295,Z 442.68,A -85,B 0,C 180,E1 -15232.612,E2 -15232.612} C_VEL
LIN {X 0,Y 320.08,Z 435.076,A -85,B 0,C 180,E1 -15236.753,E2 -15236.753} C_VEL
LIN {X 0,Y 320.84,Z 428.793,A -85,B 0,C 180,E1 -15240.255,E2 -15240.255} C_VEL
LIN {X 0,Y 321.784,Z 422.446,A -85,B 0,C 180,E1 -15243.906,E2 -15243.906} C_VEL
LIN {X 0,Y 322.334,Z 418.525,A -85,B 0,C 180,E1 -15246.222,E2 -15246.222} C_VEL
LIN {X 0,Y 322.182,Z 415.301,A -85,B 0,C 180,E1 -15248.252,E2 -15248.252} C_VEL
LIN {X 0,Y 321.23,Z 409.774,A -85,B 0,C 180,E1 -15251.938,E2 -15251.938} C_VEL
LIN {X 0,Y 320.342,Z 404.911,A -85,B 0,C 180,E1 -15255.408,E2 -15255.408} C_VEL
LIN {X 0,Y 319.565,Z 400.681,A -85,B 0,C 180,E1 -15258.717,E2 -15258.717} C_VEL
LIN {X 0,Y 319.568,Z 400.679,A -85,B 0,C 180,E1 -15262.349,E2 -15262.349} C_VEL
LIN {X 0,Y 319.567,Z 400.679,A -85,B 0,C 180,E1 -15265.124,E2 -15265.124} C_VEL
LIN {X 0,Y 319.574,Z 400.678,A -85,B 0,C 180,E1 -15269.06,E2 -15269.06} C_VEL
LIN {X 0,Y 319.613,Z 400.675,A -85,B 0,C 180,E1 -15272.498,E2 -15272.498} C_VEL
LIN {X 0,Y 319.612,Z 400.67,A -85,B 0,C 180,E1 -15275.304,E2 -15275.304} C_VEL
LIN {X 0,Y 319.604,Z 400.673,A -85,B 0,C 180,E1 -15278.048,E2 -15278.048} C_VEL
LIN {X 0,Y 319.697,Z 400.662,A -85,B 0,C 180,E1 -15280.963,E2 -15280.963} C_VEL
LIN {X 0,Y 319.738,Z 400.655,A -85,B 0,C 180,E1 -15285.276,E2 -15285.276} C_VEL
LIN {X 0,Y 319.76,Z 400.654,A -85,B 0,C 180,E1 -15289.873,E2 -15289.873} C_VEL
LIN {X 0,Y 319.919,Z 400.636,A -85,B 0,C 180,E1 -15292.426,E2 -15292.426} C_VEL
LIN {X 0,Y 319.749,Z 400.653,A -85,B 0,C 180,E1 -15294.956,E2 -15294.956} C_VEL
LIN {X 0,Y 319.995,Z 400.623,A -85,B 0,C 180,E1 -15297.482,E2 -15297.482} C_VEL
LIN {X 0,Y 320.138,Z 400.609,A -85,B 0,C 180,E1 -15300,E2 -15300} C_VEL
LIN {X 0,Y 319.995,Z 400.623,A -85,B 0,C 180,E1 -15302.517,E2 -15302.517} C_VEL
LIN {X 0,Y 319.935,Z 400.625,A -85,B 0,C 180,E1 -15306.693,E2 -15306.693} C_VEL
LIN {X 0,Y 319.765,Z 400.653,A -85,B 0,C 180,E1 -15310.127,E2 -15310.127} C_VEL
LIN {X 0,Y 319.738,Z 400.654,A -85,B 0,C 180,E1 -15314.724,E2 -15314.724} C_VEL
LIN {X 0,Y 319.696,Z 400.657,A -85,B 0,C 180,E1 -15319.037,E2 -15319.037} C_VEL
LIN {X 0,Y 319.577,Z 400.675,A -85,B 0,C 180,E1 -15323.319,E2 -15323.319} C_VEL
LIN {X 0,Y 319.641,Z 400.668,A -85,B 0,C 180,E1 -15326.087,E2 -15326.087} C_VEL
LIN {X 0,Y 319.586,Z 400.673,A -85,B 0,C 180,E1 -15328.934,E2 -15328.934} C_VEL
LIN {X 0,Y 319.537,Z 400.677,A -85,B 0,C 180,E1 -15331.861,E2 -15331.861} C_VEL
LIN {X 0,Y 319.586,Z 400.677,A -85,B 0,C 180,E1 -15335.542,E2 -15335.542} C_VEL
LIN {X 0,Y 319.565,Z 400.678,A -85,B 0,C 180,E1 -15339.668,E2 -15339.668} C_VEL
LIN {X 0,Y 319.562,Z 400.677,A -85,B 0,C 180,E1 -15343.466,E2 -15343.466} C_VEL
LIN {X 0,Y 319.567,Z 400.679,A -85,B 0,C 180,E1 -15347.017,E2 -15347.017} C_VEL
LIN {X 0,Y 319.553,Z 400.677,A -85,B 0,C 180,E1 -15350.37,E2 -15350.37} C_VEL
LIN {X 0,Y 319.586,Z 400.674,A -85,B 0,C 180,E1 -15354.456,E2 -15354.456} C_VEL
LIN {X 0,Y 319.536,Z 400.68,A -85,B 0,C 180,E1 -15358.137,E2 -15358.137} C_VEL
LIN {X 0,Y 319.616,Z 400.67,A -85,B 0,C 180,E1 -15361.589,E2 -15361.589} C_VEL
LIN {X 0,Y 319.61,Z 400.671,A -85,B 0,C 180,E1 -15365.302,E2 -15365.302} C_VEL
LIN {X 0,Y 319.603,Z 400.672,A -85,B 0,C 180,E1 -15368.046,E2 -15368.046} C_VEL
LIN {X 0,Y 319.694,Z 400.663,A -85,B 0,C 180,E1 -15370.96,E2 -15370.96} C_VEL
LIN {X 0,Y 319.734,Z 400.656,A -85,B 0,C 180,E1 -15375.275,E2 -15375.275} C_VEL
LIN {X 0,Y 319.55,Z 400.683,A -85,B 0,C 180,E1 -15378.581,E2 -15378.581} C_VEL
LIN {X 0,Y 319.296,Z 400.967,A -85,B 0,C 180,E1 -15382.093,E2 -15382.093} C_VEL
LIN {X 0,Y 319.321,Z 403.305,A -85,B 0,C 180,E1 -15384.947,E2 -15384.947} C_VEL
LIN {X 0,Y 318.689,Z 408.161,A -85,B 0,C 180,E1 -15390.471,E2 -15390.471} C_VEL
LIN {X 0,Y 318.672,Z 408.232,A -85,B 0,C 180,E1 -15390.55,E2 -15390.55} C_VEL
LIN {X 0,Y 323.358,Z 423.631,A -85,B 0,C 180,E1 -15391.617,E2 -15391.617} C_VEL
LIN {X 0,Y 326.079,Z 435.593,A -85,B 0,C 180,E1 -15392.632,E2 -15392.632} C_VEL
LIN {X 0,Y 326.95,Z 440.614,A -85,B 0,C 180,E1 -15393.115,E2 -15393.115} C_VEL
LIN {X 0,Y 325.728,Z 453.121,A -85,B 0,C 180,E1 -15394.328,E2 -15394.328} C_VEL
LIN {X 0,Y 324.49,Z 463.921,A -85,B 0,C 180,E1 -15395.666,E2 -15395.666} C_VEL
LIN {X 0,Y 323.186,Z 473.686,A -85,B 0,C 180,E1 -15397.18,E2 -15397.18} C_VEL
LIN {X 0,Y 321.992,Z 482.11,A -85,B 0,C 180,E1 -15398.786,E2 -15398.786} C_VEL
LIN {X 0,Y 320.807,Z 490.353,A -85,B 0,C 180,E1 -15400.729,E2 -15400.729} C_VEL
LIN {X 0,Y 319.86,Z 496.906,A -85,B 0,C 180,E1 -15402.69,E2 -15402.69} C_VEL
LIN {X 0,Y 319.104,Z 502.335,A -85,B 0,C 180,E1 -15404.774,E2 -15404.774} C_VEL
LIN {X 0,Y 318.617,Z 506.083,A -85,B 0,C 180,E1 -15406.661,E2 -15406.661} C_VEL
LIN {X 0,Y 318.264,Z 508.521,A -85,B 0,C 180,E1 -15408.279,E2 -15408.279} C_VEL
LIN {X 0,Y 317.948,Z 510.829,A -85,B 0,C 180,E1 -15410.709,E2 -15410.709} C_VEL
LIN {X 0,Y 317.868,Z 511.507,A -85,B 0,C 180,E1 -15412.075,E2 -15412.075} C_VEL
LIN {X 0,Y 317.842,Z 511.71,A -85,B 0,C 180,E1 -15413.451,E2 -15413.451} C_VEL
LIN {X 0,Y 317.931,Z 511.378,A -85,B 0,C 180,E1 -15414.998,E2 -15414.998} C_VEL
LIN {X 0,Y 318.079,Z 510.72,A -85,B 0,C 180,E1 -15416.222,E2 -15416.222} C_VEL
LIN {X 0,Y 318.382,Z 509.058,A -85,B 0,C 180,E1 -15417.998,E2 -15417.998} C_VEL
LIN {X 0,Y 318.992,Z 505.452,A -85,B 0,C 180,E1 -15420.443,E2 -15420.443} C_VEL
LIN {X 0,Y 319.701,Z 500.865,A -85,B 0,C 180,E1 -15422.584,E2 -15422.584} C_VEL
LIN {X 0,Y 320.727,Z 494.773,A -85,B 0,C 180,E1 -15424.728,E2 -15424.728} C_VEL
LIN {X 0,Y 321.789,Z 488.31,A -85,B 0,C 180,E1 -15426.52,E2 -15426.52} C_VEL
LIN {X 0,Y 322.974,Z 480.972,A -85,B 0,C 180,E1 -15428.171,E2 -15428.171} C_VEL
LIN {X 0,Y 324.422,Z 471.314,A -85,B 0,C 180,E1 -15429.92,E2 -15429.92} C_VEL
LIN {X 0,Y 325.922,Z 460.69,A -85,B 0,C 180,E1 -15431.456,E2 -15431.456} C_VEL
LIN {X 0,Y 327.096,Z 450.906,A -85,B 0,C 180,E1 -15432.591,E2 -15432.591} C_VEL
LIN {X 0,Y 327.915,Z 443.47,A -85,B 0,C 180,E1 -15433.297,E2 -15433.297} C_VEL
LIN {X 0,Y 327.284,Z 438.712,A -85,B 0,C 180,E1 -15433.779,E2 -15433.779} C_VEL
LIN {X 0,Y 324.341,Z 426.414,A -85,B 0,C 180,E1 -15434.932,E2 -15434.932} C_VEL
LIN {X 0,Y 320.356,Z 414.177,A -85,B 0,C 180,E1 -15435.912,E2 -15435.912} C_VEL
LIN {X 0,Y 318.872,Z 409.65,A -85,B 0,C 180,E1 -15436.225,E2 -15436.225} C_VEL
LIN {X 0,Y 319.027,Z 406.393,A -85,B 0,C 180,E1 -15440.293,E2 -15440.293} C_VEL
LIN {X 0,Y 319.173,Z 403.895,A -85,B 0,C 180,E1 -15443.521,E2 -15443.521} C_VEL
LIN {X 0,Y 319.347,Z 401.474,A -85,B 0,C 180,E1 -15446.743,E2 -15446.743} C_VEL
LIN {X 0,Y 319.396,Z 400.707,A -85,B 0,C 180,E1 -15448.123,E2 -15448.123} C_VEL
LIN {X 0,Y 319.591,Z 400.677,A -85,B 0,C 180,E1 -15451.59,E2 -15451.59} C_VEL
LIN {X 0,Y 319.605,Z 400.676,A -85,B 0,C 180,E1 -15455.038,E2 -15455.038} C_VEL
LIN {X 0,Y 318.953,Z 400.76,A -85,B 0,C 180,E1 -15456.089,E2 -15456.089} C_VEL
LIN {X 0,Y 316.109,Z 401.111,A -85,B 0,C 180,E1 -15457.801,E2 -15457.801} C_VEL
LIN {X 0,Y 313.705,Z 401.41,A -85,B 0,C 180,E1 -15459.189,E2 -15459.189} C_VEL
LIN {X 0,Y 312.694,Z 401.534,A -85,B 0,C 180,E1 -15460.263,E2 -15460.263} C_VEL
LIN {X 0,Y 312.624,Z 401.544,A -85,B 0,C 180,E1 -15460.627,E2 -15460.627} C_VEL
LIN {X 0,Y 312.681,Z 401.537,A -85,B 0,C 180,E1 -15465.112,E2 -15465.112} C_VEL
LIN {X 0,Y 312.685,Z 401.533,A -85,B 0,C 180,E1 -15469.641,E2 -15469.641} C_VEL
LIN {X 0,Y 312.854,Z 401.514,A -85,B 0,C 180,E1 -15472.254,E2 -15472.254} C_VEL
LIN {X 0,Y 312.704,Z 401.534,A -85,B 0,C 180,E1 -15474.842,E2 -15474.842} C_VEL
LIN {X 0,Y 312.976,Z 401.499,A -85,B 0,C 180,E1 -15478.713,E2 -15478.713} C_VEL
LIN {X 0,Y 313.102,Z 401.484,A -85,B 0,C 180,E1 -15480,E2 -15480} C_VEL
LIN {X 0,Y 312.942,Z 401.504,A -85,B 0,C 180,E1 -15482.574,E2 -15482.574} C_VEL
LIN {X 0,Y 312.891,Z 401.512,A -85,B 0,C 180,E1 -15486.448,E2 -15486.448} C_VEL
LIN {X 0,Y 312.769,Z 401.526,A -85,B 0,C 180,E1 -15489.05,E2 -15489.05} C_VEL
LIN {X 0,Y 312.618,Z 401.545,A -85,B 0,C 180,E1 -15492.992,E2 -15492.992} C_VEL
LIN {X 0,Y 312.62,Z 401.545,A -85,B 0,C 180,E1 -15495.651,E2 -15495.651} C_VEL
LIN {X 0,Y 312.619,Z 401.548,A -85,B 0,C 180,E1 -15499.708,E2 -15499.708} C_VEL
LIN {X 0,Y 312.584,Z 401.552,A -85,B 0,C 180,E1 -15502.815,E2 -15502.815} C_VEL
LIN {X 0,Y 312.537,Z 401.56,A -85,B 0,C 180,E1 -15506.727,E2 -15506.727} C_VEL
LIN {X 0,Y 312.522,Z 401.561,A -85,B 0,C 180,E1 -15509.653,E2 -15509.653} C_VEL
LIN {X 0,Y 312.504,Z 401.56,A -85,B 0,C 180,E1 -15513.691,E2 -15513.691} C_VEL
LIN {X 0,Y 312.538,Z 401.556,A -85,B 0,C 180,E1 -15517.384,E2 -15517.384} C_VEL
LIN {X 0,Y 312.55,Z 401.755,A -85,B 0,C 180,E1 -15519.317,E2 -15519.317} C_VEL
LIN {X 0,Y 313.168,Z 405.016,A -85,B 0,C 180,E1 -15522.319,E2 -15522.319} C_VEL
LIN {X 0,Y 313.992,Z 409.489,A -85,B 0,C 180,E1 -15526.068,E2 -15526.068} C_VEL
LIN {X 0,Y 314.794,Z 414.2,A -85,B 0,C 180,E1 -15529.655,E2 -15529.655} C_VEL
LIN {X 0,Y 315.371,Z 417.828,A -85,B 0,C 180,E1 -15532.209,E2 -15532.209} C_VEL
LIN {X 0,Y 315.175,Z 421.404,A -85,B 0,C 180,E1 -15534.57,E2 -15534.57} C_VEL
LIN {X 0,Y 314.193,Z 427.352,A -85,B 0,C 180,E1 -15538.212,E2 -15538.212} C_VEL
LIN {X 0,Y 313.277,Z 433.607,A -85,B 0,C 180,E1 -15541.897,E2 -15541.897} C_VEL
LIN {X 0,Y 312.532,Z 439.796,A -85,B 0,C 180,E1 -15545.42,E2 -15545.42} C_VEL
LIN {X 0,Y 312.372,Z 441.399,A -85,B 0,C 180,E1 -15546.233,E2 -15546.233} C_VEL
LIN {X 0,Y 315.445,Z 455.195,A -85,B 0,C 180,E1 -15547.073,E2 -15547.073} C_VEL
LIN {X 0,Y 317.125,Z 465.869,A -85,B 0,C 180,E1 -15547.871,E2 -15547.871} C_VEL
LIN {X 0,Y 318.174,Z 477.599,A -85,B 0,C 180,E1 -15548.913,E2 -15548.913} C_VEL
LIN {X 0,Y 318.666,Z 489.328,A -85,B 0,C 180,E1 -15550.182,E2 -15550.182} C_VEL
LIN {X 0,Y 316.994,Z 500.751,A -85,B 0,C 180,E1 -15551.586,E2 -15551.586} C_VEL
LIN {X 0,Y 315.456,Z 510.874,A -85,B 0,C 180,E1 -15553.167,E2 -15553.167} C_VEL
LIN {X 0,Y 314.282,Z 519.195,A -85,B 0,C 180,E1 -15554.769,E2 -15554.769} C_VEL
LIN {X 0,Y 313.01,Z 527.375,A -85,B 0,C 180,E1 -15556.697,E2 -15556.697} C_VEL
LIN {X 0,Y 312.154,Z 532.952,A -85,B 0,C 180,E1 -15558.312,E2 -15558.312} C_VEL
LIN {X 0,Y 311.52,Z 538.435,A -85,B 0,C 180,E1 -15560.261,E2 -15560.261} C_VEL
LIN {X 0,Y 311.083,Z 542.734,A -85,B 0,C 180,E1 -15562.212,E2 -15562.212} C_VEL
LIN {X 0,Y 310.905,Z 545.819,A -85,B 0,C 180,E1 -15564.057,E2 -15564.057} C_VEL
LIN {X 0,Y 310.845,Z 548.229,A -85,B 0,C 180,E1 -15566.113,E2 -15566.113} C_VEL
LIN {X 0,Y 310.853,Z 549.809,A -85,B 0,C 180,E1 -15568.707,E2 -15568.707} C_VEL
LIN {X 0,Y 310.96,Z 549.968,A -85,B 0,C 180,E1 -15570.002,E2 -15570.002} C_VEL
LIN {X 0,Y 310.885,Z 549.709,A -85,B 0,C 180,E1 -15571.298,E2 -15571.298} C_VEL
LIN {X 0,Y 310.846,Z 548.016,A -85,B 0,C 180,E1 -15573.892,E2 -15573.892} C_VEL
LIN {X 0,Y 310.904,Z 545.471,A -85,B 0,C 180,E1 -15575.942,E2 -15575.942} C_VEL
LIN {X 0,Y 311.067,Z 542.202,A -85,B 0,C 180,E1 -15577.793,E2 -15577.793} C_VEL
LIN {X 0,Y 311.524,Z 537.71,A -85,B 0,C 180,E1 -15579.744,E2 -15579.744} C_VEL
LIN {X 0,Y 312.322,Z 530.899,A -85,B 0,C 180,E1 -15582.016,E2 -15582.016} C_VEL
LIN {X 0,Y 313.427,Z 523.493,A -85,B 0,C 180,E1 -15583.951,E2 -15583.951} C_VEL
LIN {X 0,Y 314.737,Z 514.458,A -85,B 0,C 180,E1 -15585.847,E2 -15585.847} C_VEL
LIN {X 0,Y 315.896,Z 504.729,A -85,B 0,C 180,E1 -15587.481,E2 -15587.481} C_VEL
LIN {X 0,Y 317.426,Z 494.164,A -85,B 0,C 180,E1 -15588.895,E2 -15588.895} C_VEL
LIN {X 0,Y 318.187,Z 487.148,A -85,B 0,C 180,E1 -15589.686,E2 -15589.686} C_VEL
LIN {X 0,Y 317.319,Z 475.547,A -85,B 0,C 180,E1 -15590.862,E2 -15590.862} C_VEL
LIN {X 0,Y 315.909,Z 462.719,A -85,B 0,C 180,E1 -15591.907,E2 -15591.907} C_VEL
LIN {X 0,Y 313.767,Z 449.691,A -85,B 0,C 180,E1 -15592.737,E2 -15592.737} C_VEL
LIN {X 0,Y 312.286,Z 442.249,A -85,B 0,C 180,E1 -15593.121,E2 -15593.121} C_VEL
LIN {X 0,Y 313.139,Z 434.628,A -85,B 0,C 180,E1 -15597.396,E2 -15597.396} C_VEL
LIN {X 0,Y 313.915,Z 428.375,A -85,B 0,C 180,E1 -15600.995,E2 -15600.995} C_VEL
LIN {X 0,Y 314.861,Z 422.733,A -85,B 0,C 180,E1 -15604.322,E2 -15604.322} C_VEL
LIN {X 0,Y 315.336,Z 418.377,A -85,B 0,C 180,E1 -15606.998,E2 -15606.998} C_VEL
LIN {X 0,Y 314.831,Z 414.558,A -85,B 0,C 180,E1 -15609.511,E2 -15609.511} C_VEL
LIN {X 0,Y 313.903,Z 409.177,A -85,B 0,C 180,E1 -15613.269,E2 -15613.269} C_VEL
LIN {X 0,Y 313.05,Z 404.455,A -85,B 0,C 180,E1 -15616.785,E2 -15616.785} C_VEL
LIN {X 0,Y 312.513,Z 401.559,A -85,B 0,C 180,E1 -15619.188,E2 -15619.188} C_VEL
LIN {X 0,Y 312.532,Z 401.556,A -85,B 0,C 180,E1 -15622.616,E2 -15622.616} C_VEL
LIN {X 0,Y 312.527,Z 401.555,A -85,B 0,C 180,E1 -15626.312,E2 -15626.312} C_VEL
LIN {X 0,Y 312.545,Z 401.554,A -85,B 0,C 180,E1 -15630.35,E2 -15630.35} C_VEL
LIN {X 0,Y 312.604,Z 401.544,A -85,B 0,C 180,E1 -15634.067,E2 -15634.067} C_VEL
LIN {X 0,Y 312.595,Z 401.544,A -85,B 0,C 180,E1 -15637.529,E2 -15637.529} C_VEL
LIN {X 0,Y 312.646,Z 401.539,A -85,B 0,C 180,E1 -15641.657,E2 -15641.657} C_VEL
LIN {X 0,Y 312.701,Z 401.532,A -85,B 0,C 180,E1 -15645.686,E2 -15645.686} C_VEL
LIN {X 0,Y 312.706,Z 401.532,A -85,B 0,C 180,E1 -15649.642,E2 -15649.642} C_VEL
LIN {X 0,Y 312.86,Z 401.517,A -85,B 0,C 180,E1 -15652.254,E2 -15652.254} C_VEL
LIN {X 0,Y 312.719,Z 401.529,A -85,B 0,C 180,E1 -15654.842,E2 -15654.842} C_VEL
LIN {X 0,Y 312.995,Z 401.495,A -85,B 0,C 180,E1 -15658.713,E2 -15658.713} C_VEL
LIN {X 0,Y 312.995,Z 401.494,A -85,B 0,C 180,E1 -15661.287,E2 -15661.287} C_VEL
LIN {X 0,Y 312.721,Z 401.525,A -85,B 0,C 180,E1 -15665.157,E2 -15665.157} C_VEL
LIN {X 0,Y 312.879,Z 401.506,A -85,B 0,C 180,E1 -15667.745,E2 -15667.745} C_VEL
LIN {X 0,Y 312.676,Z 401.537,A -85,B 0,C 180,E1 -15671.671,E2 -15671.671} C_VEL
LIN {X 0,Y 312.707,Z 401.53,A -85,B 0,C 180,E1 -15674.887,E2 -15674.887} C_VEL
LIN {X 0,Y 312.637,Z 401.536,A -85,B 0,C 180,E1 -15679.236,E2 -15679.236} C_VEL
LIN {X 0,Y 312.553,Z 401.547,A -85,B 0,C 180,E1 -15682.788,E2 -15682.788} C_VEL
LIN {X 0,Y 312.609,Z 401.545,A -85,B 0,C 180,E1 -15685.935,E2 -15685.935} C_VEL
LIN {X 0,Y 312.545,Z 401.552,A -85,B 0,C 180,E1 -15689.65,E2 -15689.65} C_VEL
LIN {X 0,Y 312.526,Z 401.553,A -85,B 0,C 180,E1 -15693.688,E2 -15693.688} C_VEL
LIN {X 0,Y 312.527,Z 401.558,A -85,B 0,C 180,E1 -15697.385,E2 -15697.385} C_VEL
LIN {X 0,Y 312.497,Z 401.557,A -85,B 0,C 180,E1 -15700.708,E2 -15700.708} C_VEL
LIN {X 0,Y 312.478,Z 401.555,A -85,B 0,C 180,E1 -15704.205,E2 -15704.205} C_VEL
LIN {X 0,Y 312.492,Z 401.557,A -85,B 0,C 180,E1 -15707.917,E2 -15707.917} C_VEL
LIN {X 0,Y 312.504,Z 401.559,A -85,B 0,C 180,E1 -15710.97,E2 -15710.97} C_VEL
LIN {X 0,Y 312.538,Z 401.55,A -85,B 0,C 180,E1 -15714.219,E2 -15714.219} C_VEL
LIN {X 0,Y 312.509,Z 401.557,A -85,B 0,C 180,E1 -15717.332,E2 -15717.332} C_VEL
LIN {X 0,Y 312.55,Z 401.552,A -85,B 0,C 180,E1 -15721.277,E2 -15721.277} C_VEL
LIN {X 0,Y 312.591,Z 401.55,A -85,B 0,C 180,E1 -15724.709,E2 -15724.709} C_VEL
LIN {X 0,Y 312.593,Z 401.545,A -85,B 0,C 180,E1 -15727.527,E2 -15727.527} C_VEL
LIN {X 0,Y 312.643,Z 401.538,A -85,B 0,C 180,E1 -15731.654,E2 -15731.654} C_VEL
LIN {X 0,Y 312.69,Z 401.533,A -85,B 0,C 180,E1 -15735.684,E2 -15735.684} C_VEL
LIN {X 0,Y 312.425,Z 401.566,A -85,B 0,C 180,E1 -15739.63,E2 -15739.63} C_VEL
LIN {X 0,Y 312.263,Z 401.857,A -85,B 0,C 180,E1 -15742.01,E2 -15742.01} C_VEL
LIN {X 0,Y 312.294,Z 404.133,A -85,B 0,C 180,E1 -15744.833,E2 -15744.833} C_VEL
LIN {X 0,Y 311.646,Z 408.709,A -85,B 0,C 180,E1 -15750.078,E2 -15750.078} C_VEL
LIN {X 0,Y 315.463,Z 421.105,A -85,B 0,C 180,E1 -15750.921,E2 -15750.921} C_VEL
LIN {X 0,Y 318.167,Z 431.456,A -85,B 0,C 180,E1 -15751.778,E2 -15751.778} C_VEL
LIN {X 0,Y 320.207,Z 441.747,A -85,B 0,C 180,E1 -15752.776,E2 -15752.776} C_VEL
LIN {X 0,Y 318.982,Z 453.514,A -85,B 0,C 180,E1 -15753.946,E2 -15753.946} C_VEL
LIN {X 0,Y 317.65,Z 464.678,A -85,B 0,C 180,E1 -15755.362,E2 -15755.362} C_VEL
LIN {X 0,Y 316.21,Z 475.006,A -85,B 0,C 180,E1 -15757.019,E2 -15757.019} C_VEL
LIN {X 0,Y 314.97,Z 483.291,A -85,B 0,C 180,E1 -15758.66,E2 -15758.66} C_VEL
LIN {X 0,Y 313.769,Z 491.366,A -85,B 0,C 180,E1 -15760.646,E2 -15760.646} C_VEL
LIN {X 0,Y 312.951,Z 496.846,A -85,B 0,C 180,E1 -15762.316,E2 -15762.316} C_VEL
LIN {X 0,Y 312.116,Z 502.456,A -85,B 0,C 180,E1 -15764.478,E2 -15764.478} C_VEL
LIN {X 0,Y 311.612,Z 506.225,A -85,B 0,C 180,E1 -15766.372,E2 -15766.372} C_VEL
LIN {X 0,Y 311.163,Z 509.23,A -85,B 0,C 180,E1 -15768.446,E2 -15768.446} C_VEL
LIN {X 0,Y 310.944,Z 510.619,A -85,B 0,C 180,E1 -15769.815,E2 -15769.815} C_VEL
LIN {X 0,Y 310.788,Z 511.91,A -85,B 0,C 180,E1 -15772.005,E2 -15772.005} C_VEL
LIN {X 0,Y 310.775,Z 512.094,A -85,B 0,C 180,E1 -15774.017,E2 -15774.017} C_VEL
LIN {X 0,Y 310.897,Z 511.676,A -85,B 0,C 180,E1 -15775.433,E2 -15775.433} C_VEL
LIN {X 0,Y 311.091,Z 510.734,A -85,B 0,C 180,E1 -15776.858,E2 -15776.858} C_VEL
LIN {X 0,Y 311.378,Z 509.292,A -85,B 0,C 180,E1 -15778.327,E2 -15778.327} C_VEL
LIN {X 0,Y 311.924,Z 506.233,A -85,B 0,C 180,E1 -15780.45,E2 -15780.45} C_VEL
LIN {X 0,Y 312.651,Z 501.752,A -85,B 0,C 180,E1 -15782.645,E2 -15782.645} C_VEL
LIN {X 0,Y 313.704,Z 495.782,A -85,B 0,C 180,E1 -15784.836,E2 -15784.836} C_VEL
LIN {X 0,Y 314.828,Z 489.338,A -85,B 0,C 180,E1 -15786.696,E2 -15786.696} C_VEL
LIN {X 0,Y 316.135,Z 481.634,A -85,B 0,C 180,E1 -15788.492,E2 -15788.492} C_VEL
LIN {X 0,Y 317.518,Z 472.893,A -85,B 0,C 180,E1 -15790.136,E2 -15790.136} C_VEL
LIN {X 0,Y 318.947,Z 463.504,A -85,B 0,C 180,E1 -15791.565,E2 -15791.565} C_VEL
LIN {X 0,Y 320.43,Z 451.847,A -85,B 0,C 180,E1 -15792.99,E2 -15792.99} C_VEL
LIN {X 0,Y 321.262,Z 443.744,A -85,B 0,C 180,E1 -15793.787,E2 -15793.787} C_VEL
LIN {X 0,Y 319.001,Z 432.815,A -85,B 0,C 180,E1 -15794.92,E2 -15794.92} C_VEL
LIN {X 0,Y 315.561,Z 420.715,A -85,B 0,C 180,E1 -15796.009,E2 -15796.009} C_VEL
LIN {X 0,Y 311.911,Z 410.552,A -85,B 0,C 180,E1 -15796.797,E2 -15796.797} C_VEL
LIN {X 0,Y 311.857,Z 410.089,A -85,B 0,C 180,E1 -15796.863,E2 -15796.863} C_VEL
LIN {X 0,Y 312.024,Z 406.936,A -85,B 0,C 180,E1 -15800.901,E2 -15800.901} C_VEL
LIN {X 0,Y 312.183,Z 404.455,A -85,B 0,C 180,E1 -15804.174,E2 -15804.174} C_VEL
LIN {X 0,Y 312.329,Z 402.168,A -85,B 0,C 180,E1 -15807.313,E2 -15807.313} C_VEL
LIN {X 0,Y 312.418,Z 401.575,A -85,B 0,C 180,E1 -15808.842,E2 -15808.842} C_VEL
LIN {X 0,Y 312.551,Z 401.554,A -85,B 0,C 180,E1 -15811.823,E2 -15811.823} C_VEL
LIN {X 0,Y 312.56,Z 401.552,A -85,B 0,C 180,E1 -15815.028,E2 -15815.028} C_VEL
LIN {X 0,Y 312.614,Z 401.547,A -85,B 0,C 180,E1 -15817.531,E2 -15817.531} C_VEL
LIN {X 0,Y 312.624,Z 401.544,A -85,B 0,C 180,E1 -15820.627,E2 -15820.627} C_VEL
LIN {X 0,Y 311.986,Z 401.627,A -85,B 0,C 180,E1 -15821.702,E2 -15821.702} C_VEL
LIN {X 0,Y 309.14,Z 401.98,A -85,B 0,C 180,E1 -15823.453,E2 -15823.453} C_VEL
LIN {X 0,Y 306.706,Z 402.28,A -85,B 0,C 180,E1 -15824.872,E2 -15824.872} C_VEL
LIN {X 0,Y 305.657,Z 402.412,A -85,B 0,C 180,E1 -15825.972,E2 -15825.972} C_VEL
LIN {X 0,Y 305.571,Z 402.418,A -85,B 0,C 180,E1 -15826.344,E2 -15826.344} C_VEL
LIN {X 0,Y 305.778,Z 402.397,A -85,B 0,C 180,E1 -15831.207,E2 -15831.207} C_VEL
LIN {X 0,Y 305.836,Z 402.385,A -85,B 0,C 180,E1 -15833.402,E2 -15833.402} C_VEL
LIN {X 0,Y 305.942,Z 402.375,A -85,B 0,C 180,E1 -15838.684,E2 -15838.684} C_VEL
LIN {X 0,Y 305.943,Z 402.376,A -85,B 0,C 180,E1 -15841.316,E2 -15841.316} C_VEL
LIN {X 0,Y 305.674,Z 402.409,A -85,B 0,C 180,E1 -15845.277,E2 -15845.277} C_VEL
LIN {X 0,Y 305.794,Z 402.395,A -85,B 0,C 180,E1 -15847.926,E2 -15847.926} C_VEL
LIN {X 0,Y 305.587,Z 402.421,A -85,B 0,C 180,E1 -15851.946,E2 -15851.946} C_VEL
LIN {X 0,Y 305.62,Z 402.417,A -85,B 0,C 180,E1 -15855.036,E2 -15855.036} C_VEL
LIN {X 0,Y 305.597,Z 402.421,A -85,B 0,C 180,E1 -15859.466,E2 -15859.466} C_VEL
LIN {X 0,Y 305.539,Z 402.43,A -85,B 0,C 180,E1 -15863.072,E2 -15863.072} C_VEL
LIN {X 0,Y 305.517,Z 402.433,A -85,B 0,C 180,E1 -15866.223,E2 -15866.223} C_VEL
LIN {X 0,Y 305.472,Z 402.439,A -85,B 0,C 180,E1 -15869.049,E2 -15869.049} C_VEL
LIN {X 0,Y 305.427,Z 402.444,A -85,B 0,C 180,E1 -15871.954,E2 -15871.954} C_VEL
LIN {X 0,Y 305.448,Z 402.44,A -85,B 0,C 180,E1 -15875.115,E2 -15875.115} C_VEL
LIN {X 0,Y 305.522,Z 402.566,A -85,B 0,C 180,E1 -15878.551,E2 -15878.551} C_VEL
LIN {X 0,Y 306.108,Z 405.901,A -85,B 0,C 180,E1 -15881.745,E2 -15881.745} C_VEL
LIN {X 0,Y 306.814,Z 409.911,A -85,B 0,C 180,E1 -15885.243,E2 -15885.243} C_VEL
LIN {X 0,Y 307.669,Z 414.548,A -85,B 0,C 180,E1 -15888.922,E2 -15888.922} C_VEL
LIN {X 0,Y 308.351,Z 418.758,A -85,B 0,C 180,E1 -15892.024,E2 -15892.024} C_VEL
LIN {X 0,Y 308.305,Z 421.152,A -85,B 0,C 180,E1 -15893.656,E2 -15893.656} C_VEL
LIN {X 0,Y 307.543,Z 425.966,A -85,B 0,C 180,E1 -15896.743,E2 -15896.743} C_VEL
LIN {X 0,Y 306.533,Z 432.268,A -85,B 0,C 180,E1 -15900.604,E2 -15900.604} C_VEL
LIN {X 0,Y 305.729,Z 438.2,A -85,B 0,C 180,E1 -15904.106,E2 -15904.106} C_VEL
LIN {X 0,Y 305.417,Z 440.75,A -85,B 0,C 180,E1 -15905.588,E2 -15905.588} C_VEL
LIN {X 0,Y 308.576,Z 454.854,A -85,B 0,C 180,E1 -15906.492,E2 -15906.492} C_VEL
LIN {X 0,Y 310.554,Z 467.63,A -85,B 0,C 180,E1 -15907.508,E2 -15907.508} C_VEL
LIN {X 0,Y 311.517,Z 480.331,A -85,B 0,C 180,E1 -15908.715,E2 -15908.715} C_VEL
LIN {X 0,Y 311.796,Z 490.63,A -85,B 0,C 180,E1 -15909.898,E2 -15909.898} C_VEL
LIN {X 0,Y 310.064,Z 501.645,A -85,B 0,C 180,E1 -15911.33,E2 -15911.33} C_VEL
LIN {X 0,Y 308.428,Z 511.919,A -85,B 0,C 180,E1 -15913.017,E2 -15913.017} C_VEL
LIN {X 0,Y 307.144,Z 520.414,A -85,B 0,C 180,E1 -15914.746,E2 -15914.746} C_VEL
LIN {X 0,Y 305.869,Z 528.259,A -85,B 0,C 180,E1 -15916.719,E2 -15916.719} C_VEL
LIN {X 0,Y 304.924,Z 534.572,A -85,B 0,C 180,E1 -15918.705,E2 -15918.705} C_VEL
LIN {X 0,Y 304.306,Z 539.618,A -85,B 0,C 180,E1 -15920.699,E2 -15920.699} C_VEL
LIN {X 0,Y 303.946,Z 543.541,A -85,B 0,C 180,E1 -15922.696,E2 -15922.696} C_VEL
LIN {X 0,Y 303.769,Z 546.437,A -85,B 0,C 180,E1 -15924.693,E2 -15924.693} C_VEL
LIN {X 0,Y 303.754,Z 547.819,A -85,B 0,C 180,E1 -15926.022,E2 -15926.022} C_VEL
LIN {X 0,Y 303.76,Z 549.384,A -85,B 0,C 180,E1 -15928.677,E2 -15928.677} C_VEL
LIN {X 0,Y 303.872,Z 549.532,A -85,B 0,C 180,E1 -15930.003,E2 -15930.003} C_VEL
LIN {X 0,Y 303.792,Z 549.267,A -85,B 0,C 180,E1 -15931.328,E2 -15931.328} C_VEL
LIN {X 0,Y 303.778,Z 547.559,A -85,B 0,C 180,E1 -15933.982,E2 -15933.982} C_VEL
LIN {X 0,Y 303.833,Z 545.203,A -85,B 0,C 180,E1 -15935.932,E2 -15935.932} C_VEL
LIN {X 0,Y 304.019,Z 541.715,A -85,B 0,C 180,E1 -15937.975,E2 -15937.975} C_VEL
LIN {X 0,Y 304.483,Z 537.204,A -85,B 0,C 180,E1 -15939.971,E2 -15939.971} C_VEL
LIN {X 0,Y 305.342,Z 530.365,A -85,B 0,C 180,E1 -15942.295,E2 -15942.295} C_VEL
LIN {X 0,Y 306.471,Z 522.935,A -85,B 0,C 180,E1 -15944.274,E2 -15944.274} C_VEL
LIN {X 0,Y 307.789,Z 514.307,A -85,B 0,C 180,E1 -15946.126,E2 -15946.126} C_VEL
LIN {X 0,Y 308.93,Z 505.173,A -85,B 0,C 180,E1 -15947.717,E2 -15947.717} C_VEL
LIN {X 0,Y 310.514,Z 494.789,A -85,B 0,C 180,E1 -15949.161,E2 -15949.161} C_VEL
LIN {X 0,Y 311.284,Z 487.925,A -85,B 0,C 180,E1 -15949.97,E2 -15949.97} C_VEL
LIN {X 0,Y 310.455,Z 475.929,A -85,B 0,C 180,E1 -15951.238,E2 -15951.238} C_VEL
LIN {X 0,Y 309.139,Z 463.389,A -85,B 0,C 180,E1 -15952.297,E2 -15952.297} C_VEL
LIN {X 0,Y 306.915,Z 450.106,A -85,B 0,C 180,E1 -15953.194,E2 -15953.194} C_VEL
LIN {X 0,Y 305.3,Z 441.847,A -85,B 0,C 180,E1 -15953.634,E2 -15953.634} C_VEL
LIN {X 0,Y 306.044,Z 435.416,A -85,B 0,C 180,E1 -15957.343,E2 -15957.343} C_VEL
LIN {X 0,Y 306.855,Z 429.166,A -85,B 0,C 180,E1 -15961.021,E2 -15961.021} C_VEL
LIN {X 0,Y 307.915,Z 422.952,A -85,B 0,C 180,E1 -15964.795,E2 -15964.795} C_VEL
LIN {X 0,Y 308.306,Z 419.329,A -85,B 0,C 180,E1 -15967.075,E2 -15967.075} C_VEL
LIN {X 0,Y 307.757,Z 415.394,A -85,B 0,C 180,E1 -15969.75,E2 -15969.75} C_VEL
LIN {X 0,Y 306.908,Z 410.288,A -85,B 0,C 180,E1 -15973.394,E2 -15973.394} C_VEL
LIN {X 0,Y 305.96,Z 405.192,A -85,B 0,C 180,E1 -15977.314,E2 -15977.314} C_VEL
LIN {X 0,Y 305.482,Z 402.435,A -85,B 0,C 180,E1 -15979.642,E2 -15979.642} C_VEL
LIN {X 0,Y 305.488,Z 402.431,A -85,B 0,C 180,E1 -15983.632,E2 -15983.632} C_VEL
LIN {X 0,Y 305.473,Z 402.435,A -85,B 0,C 180,E1 -15986.484,E2 -15986.484} C_VEL
LIN {X 0,Y 305.465,Z 402.434,A -85,B 0,C 180,E1 -15989.591,E2 -15989.591} C_VEL
LIN {X 0,Y 305.522,Z 402.43,A -85,B 0,C 180,E1 -15992.608,E2 -15992.608} C_VEL
LIN {X 0,Y 305.515,Z 402.426,A -85,B 0,C 180,E1 -15995.539,E2 -15995.539} C_VEL
LIN {X 0,Y 305.527,Z 402.426,A -85,B 0,C 180,E1 -15999.815,E2 -15999.815} C_VEL
LIN {X 0,Y 305.582,Z 402.423,A -85,B 0,C 180,E1 -16002.603,E2 -16002.603} C_VEL
LIN {X 0,Y 305.657,Z 402.41,A -85,B 0,C 180,E1 -16005.349,E2 -16005.349} C_VEL
LIN {X 0,Y 305.643,Z 402.411,A -85,B 0,C 180,E1 -16009.4,E2 -16009.4} C_VEL
LIN {X 0,Y 305.804,Z 402.395,A -85,B 0,C 180,E1 -16012.074,E2 -16012.074} C_VEL
LIN {X 0,Y 305.691,Z 402.406,A -85,B 0,C 180,E1 -16014.723,E2 -16014.723} C_VEL
LIN {X 0,Y 305.962,Z 402.371,A -85,B 0,C 180,E1 -16018.684,E2 -16018.684} C_VEL
LIN {X 0,Y 305.962,Z 402.371,A -85,B 0,C 180,E1 -16021.316,E2 -16021.316} C_VEL
LIN {X 0,Y 305.858,Z 402.376,A -85,B 0,C 180,E1 -16026.597,E2 -16026.597} C_VEL
LIN {X 0,Y 305.743,Z 402.394,A -85,B 0,C 180,E1 -16029.259,E2 -16029.259} C_VEL
LIN {X 0,Y 305.595,Z 402.417,A -85,B 0,C 180,E1 -16033.296,E2 -16033.296} C_VEL
LIN {X 0,Y 305.601,Z 402.416,A -85,B 0,C 180,E1 -16036.02,E2 -16036.02} C_VEL
LIN {X 0,Y 305.584,Z 402.415,A -85,B 0,C 180,E1 -16039.444,E2 -16039.444} C_VEL
LIN {X 0,Y 305.497,Z 402.426,A -85,B 0,C 180,E1 -16043.04,E2 -16043.04} C_VEL
LIN {X 0,Y 305.538,Z 402.424,A -85,B 0,C 180,E1 -16046.22,E2 -16046.22} C_VEL
LIN {X 0,Y 305.495,Z 402.429,A -85,B 0,C 180,E1 -16049.046,E2 -16049.046} C_VEL
LIN {X 0,Y 305.449,Z 402.429,A -85,B 0,C 180,E1 -16051.951,E2 -16051.951} C_VEL
LIN {X 0,Y 305.469,Z 402.431,A -85,B 0,C 180,E1 -16055.112,E2 -16055.112} C_VEL
LIN {X 0,Y 305.447,Z 402.435,A -85,B 0,C 180,E1 -16058.525,E2 -16058.525} C_VEL
LIN {X 0,Y 305.465,Z 402.43,A -85,B 0,C 180,E1 -16062.585,E2 -16062.585} C_VEL
LIN {X 0,Y 305.449,Z 402.433,A -85,B 0,C 180,E1 -16066.347,E2 -16066.347} C_VEL
LIN {X 0,Y 305.464,Z 402.432,A -85,B 0,C 180,E1 -16069.891,E2 -16069.891} C_VEL
LIN {X 0,Y 305.486,Z 402.429,A -85,B 0,C 180,E1 -16073.63,E2 -16073.63} C_VEL
LIN {X 0,Y 305.471,Z 402.434,A -85,B 0,C 180,E1 -16076.482,E2 -16076.482} C_VEL
LIN {X 0,Y 305.463,Z 402.431,A -85,B 0,C 180,E1 -16079.589,E2 -16079.589} C_VEL
LIN {X 0,Y 305.52,Z 402.429,A -85,B 0,C 180,E1 -16082.606,E2 -16082.606} C_VEL
LIN {X 0,Y 305.513,Z 402.426,A -85,B 0,C 180,E1 -16085.537,E2 -16085.537} C_VEL
LIN {X 0,Y 305.525,Z 402.425,A -85,B 0,C 180,E1 -16089.813,E2 -16089.813} C_VEL
LIN {X 0,Y 305.579,Z 402.422,A -85,B 0,C 180,E1 -16092.601,E2 -16092.601} C_VEL
LIN {X 0,Y 305.649,Z 402.41,A -85,B 0,C 180,E1 -16095.347,E2 -16095.347} C_VEL
LIN {X 0,Y 305.387,Z 402.443,A -85,B 0,C 180,E1 -16099.389,E2 -16099.389} C_VEL
LIN {X 0,Y 305.221,Z 402.839,A -85,B 0,C 180,E1 -16102.056,E2 -16102.056} C_VEL
LIN {X 0,Y 305.269,Z 404.982,A -85,B 0,C 180,E1 -16104.714,E2 -16104.714} C_VEL
LIN {X 0,Y 304.613,Z 409.045,A -85,B 0,C 180,E1 -16109.543,E2 -16109.543} C_VEL
LIN {X 0,Y 308.988,Z 423.315,A -85,B 0,C 180,E1 -16110.577,E2 -16110.577} C_VEL
LIN {X 0,Y 311.582,Z 433.519,A -85,B 0,C 180,E1 -16111.473,E2 -16111.473} C_VEL
LIN {X 0,Y 313.395,Z 443.356,A -85,B 0,C 180,E1 -16112.467,E2 -16112.467} C_VEL
LIN {X 0,Y 312.089,Z 455.32,A -85,B 0,C 180,E1 -16113.71,E2 -16113.71} C_VEL
LIN {X 0,Y 310.683,Z 466.366,A -85,B 0,C 180,E1 -16115.189,E2 -16115.189} C_VEL
LIN {X 0,Y 309.246,Z 476.31,A -85,B 0,C 180,E1 -16116.85,E2 -16116.85} C_VEL
LIN {X 0,Y 307.98,Z 484.452,A -85,B 0,C 180,E1 -16118.527,E2 -16118.527} C_VEL
LIN {X 0,Y 306.737,Z 492.353,A -85,B 0,C 180,E1 -16120.559,E2 -16120.559} C_VEL
LIN {X 0,Y 305.728,Z 498.686,A -85,B 0,C 180,E1 -16122.611,E2 -16122.611} C_VEL
LIN {X 0,Y 305.007,Z 503.679,A -85,B 0,C 180,E1 -16124.68,E2 -16124.68} C_VEL
LIN {X 0,Y 304.428,Z 507.501,A -85,B 0,C 180,E1 -16126.77,E2 -16126.77} C_VEL
LIN {X 0,Y 304.009,Z 510.229,A -85,B 0,C 180,E1 -16128.881,E2 -16128.881} C_VEL
LIN {X 0,Y 303.827,Z 511.468,A -85,B 0,C 180,E1 -16130.299,E2 -16130.299} C_VEL
LIN {X 0,Y 303.691,Z 512.425,A -85,B 0,C 180,E1 -16132.229,E2 -16132.229} C_VEL
LIN {X 0,Y 303.749,Z 512.428,A -85,B 0,C 180,E1 -16134.609,E2 -16134.609} C_VEL
LIN {X 0,Y 303.892,Z 511.803,A -85,B 0,C 180,E1 -16136.063,E2 -16136.063} C_VEL
LIN {X 0,Y 304.119,Z 510.728,A -85,B 0,C 180,E1 -16137.525,E2 -16137.525} C_VEL
LIN {X 0,Y 304.668,Z 508.119,A -85,B 0,C 180,E1 -16139.729,E2 -16139.729} C_VEL
LIN {X 0,Y 305.306,Z 504.225,A -85,B 0,C 180,E1 -16141.965,E2 -16141.965} C_VEL
LIN {X 0,Y 306.372,Z 498.577,A -85,B 0,C 180,E1 -16144.328,E2 -16144.328} C_VEL
LIN {X 0,Y 307.578,Z 491.985,A -85,B 0,C 180,E1 -16146.443,E2 -16146.443} C_VEL
LIN {X 0,Y 308.924,Z 484.621,A -85,B 0,C 180,E1 -16148.307,E2 -16148.307} C_VEL
LIN {X 0,Y 310.372,Z 475.846,A -85,B 0,C 180,E1 -16150.103,E2 -16150.103} C_VEL
LIN {X 0,Y 312.052,Z 465.72,A -85,B 0,C 180,E1 -16151.76,E2 -16151.76} C_VEL
LIN {X 0,Y 313.507,Z 455.187,A -85,B 0,C 180,E1 -16153.131,E2 -16153.131} C_VEL
LIN {X 0,Y 314.623,Z 445.848,A -85,B 0,C 180,E1 -16154.118,E2 -16154.118} C_VEL
LIN {X 0,Y 312.816,Z 435.997,A -85,B 0,C 180,E1 -16155.196,E2 -16155.196} C_VEL
LIN {X 0,Y 309.7,Z 424.635,A -85,B 0,C 180,E1 -16156.297,E2 -16156.297} C_VEL
LIN {X 0,Y 305.565,Z 413.103,A -85,B 0,C 180,E1 -16157.279,E2 -16157.279} C_VEL
LIN {X 0,Y 304.831,Z 410.573,A -85,B 0,C 180,E1 -16157.484,E2 -16157.484} C_VEL
LIN {X 0,Y 305.043,Z 407.463,A -85,B 0,C 180,E1 -16161.562,E2 -16161.562} C_VEL
LIN {X 0,Y 305.182,Z 405.044,A -85,B 0,C 180,E1 -16164.85,E2 -16164.85} C_VEL
LIN {X 0,Y 305.329,Z 402.543,A -85,B 0,C 180,E1 -16168.386,E2 -16168.386} C_VEL
LIN {X 0,Y 305.479,Z 402.435,A -85,B 0,C 180,E1 -16171.11,E2 -16171.11} C_VEL
LIN {X 0,Y 305.556,Z 402.427,A -85,B 0,C 180,E1 -16174.087,E2 -16174.087} C_VEL
LIN {X 0,Y 305.544,Z 402.427,A -85,B 0,C 180,E1 -16178.406,E2 -16178.406} C_VEL
LIN {X 0,Y 305.583,Z 402.421,A -85,B 0,C 180,E1 -16181.217,E2 -16181.217} C_VEL
LIN {X 0,Y 305.63,Z 402.415,A -85,B 0,C 180,E1 -16185.348,E2 -16185.348} C_VEL
LIN {X 0,Y 305.571,Z 402.418,A -85,B 0,C 180,E1 -16186.344,E2 -16186.344} C_VEL
LIN {X 0,Y 304.921,Z 402.502,A -85,B 0,C 180,E1 -16187.444,E2 -16187.444} C_VEL
LIN {X 0,Y 302.155,Z 402.852,A -85,B 0,C 180,E1 -16189.238,E2 -16189.238} C_VEL
LIN {X 0,Y 299.815,Z 403.144,A -85,B 0,C 180,E1 -16190.692,E2 -16190.692} C_VEL
LIN {X 0,Y 298.815,Z 403.264,A -85,B 0,C 180,E1 -16191.817,E2 -16191.817} C_VEL
LIN {X 0,Y 298.735,Z 403.271,A -85,B 0,C 180,E1 -16192.197,E2 -16192.197} C_VEL
LIN {X 0,Y 298.646,Z 403.286,A -85,B 0,C 180,E1 -16194.599,E2 -16194.599} C_VEL
LIN {X 0,Y 298.908,Z 403.251,A -85,B 0,C 180,E1 -16198.653,E2 -16198.653} C_VEL
LIN {X 0,Y 298.91,Z 403.252,A -85,B 0,C 180,E1 -16201.347,E2 -16201.347} C_VEL
LIN {X 0,Y 298.645,Z 403.285,A -85,B 0,C 180,E1 -16205.401,E2 -16205.401} C_VEL
LIN {X 0,Y 298.739,Z 403.274,A -85,B 0,C 180,E1 -16208.115,E2 -16208.115} C_VEL
LIN {X 0,Y 298.537,Z 403.298,A -85,B 0,C 180,E1 -16212.232,E2 -16212.232} C_VEL
LIN {X 0,Y 298.588,Z 403.293,A -85,B 0,C 180,E1 -16215.21,E2 -16215.21} C_VEL
LIN {X 0,Y 298.549,Z 403.3,A -85,B 0,C 180,E1 -16219.685,E2 -16219.685} C_VEL
LIN {X 0,Y 298.473,Z 403.31,A -85,B 0,C 180,E1 -16223.597,E2 -16223.597} C_VEL
LIN {X 0,Y 298.471,Z 403.312,A -85,B 0,C 180,E1 -16226.576,E2 -16226.576} C_VEL
LIN {X 0,Y 298.401,Z 403.32,A -85,B 0,C 180,E1 -16229.643,E2 -16229.643} C_VEL
LIN {X 0,Y 298.38,Z 403.321,A -85,B 0,C 180,E1 -16232.802,E2 -16232.802} C_VEL
LIN {X 0,Y 298.456,Z 403.309,A -85,B 0,C 180,E1 -16236.816,E2 -16236.816} C_VEL
LIN {X 0,Y 298.436,Z 403.402,A -85,B 0,C 180,E1 -16237.755,E2 -16237.755} C_VEL
LIN {X 0,Y 299.082,Z 406.893,A -85,B 0,C 180,E1 -16241.245,E2 -16241.245} C_VEL
LIN {X 0,Y 299.744,Z 410.711,A -85,B 0,C 180,E1 -16244.701,E2 -16244.701} C_VEL
LIN {X 0,Y 300.585,Z 415.236,A -85,B 0,C 180,E1 -16248.435,E2 -16248.435} C_VEL
LIN {X 0,Y 301.313,Z 419.618,A -85,B 0,C 180,E1 -16251.777,E2 -16251.777} C_VEL
LIN {X 0,Y 301.303,Z 422.082,A -85,B 0,C 180,E1 -16253.506,E2 -16253.506} C_VEL
LIN {X 0,Y 300.528,Z 426.885,A -85,B 0,C 180,E1 -16256.668,E2 -16256.668} C_VEL
LIN {X 0,Y 299.506,Z 432.95,A -85,B 0,C 180,E1 -16260.481,E2 -16260.481} C_VEL
LIN {X 0,Y 298.65,Z 439.063,A -85,B 0,C 180,E1 -16264.196,E2 -16264.196} C_VEL
LIN {X 0,Y 298.46,Z 440.292,A -85,B 0,C 180,E1 -16264.925,E2 -16264.925} C_VEL
LIN {X 0,Y 301.662,Z 454.17,A -85,B 0,C 180,E1 -16265.85,E2 -16265.85} C_VEL
LIN {X 0,Y 303.641,Z 466.148,A -85,B 0,C 180,E1 -16266.832,E2 -16266.832} C_VEL
LIN {X 0,Y 304.602,Z 477.866,A -85,B 0,C 180,E1 -16267.958,E2 -16267.958} C_VEL
LIN {X 0,Y 305.101,Z 490.506,A -85,B 0,C 180,E1 -16269.437,E2 -16269.437} C_VEL
LIN {X 0,Y 303.35,Z 501.442,A -85,B 0,C 180,E1 -16270.901,E2 -16270.901} C_VEL
LIN {X 0,Y 301.556,Z 512.029,A -85,B 0,C 180,E1 -16272.687,E2 -16272.687} C_VEL
LIN {X 0,Y 300.284,Z 520.139,A -85,B 0,C 180,E1 -16274.389,E2 -16274.389} C_VEL
LIN {X 0,Y 298.928,Z 527.943,A -85,B 0,C 180,E1 -16276.405,E2 -16276.405} C_VEL
LIN {X 0,Y 297.917,Z 534.232,A -85,B 0,C 180,E1 -16278.436,E2 -16278.436} C_VEL
LIN {X 0,Y 297.27,Z 539.258,A -85,B 0,C 180,E1 -16280.477,E2 -16280.477} C_VEL
LIN {X 0,Y 296.865,Z 543.159,A -85,B 0,C 180,E1 -16282.521,E2 -16282.521} C_VEL
LIN {X 0,Y 296.688,Z 546.037,A -85,B 0,C 180,E1 -16284.566,E2 -16284.566} C_VEL
LIN {X 0,Y 296.667,Z 547.411,A -85,B 0,C 180,E1 -16285.927,E2 -16285.927} C_VEL
LIN {X 0,Y 296.632,Z 548.385,A -85,B 0,C 180,E1 -16287.287,E2 -16287.287} C_VEL
LIN {X 0,Y 296.669,Z 548.959,A -85,B 0,C 180,E1 -16288.645,E2 -16288.645} C_VEL
LIN {X 0,Y 296.783,Z 549.096,A -85,B 0,C 180,E1 -16290.003,E2 -16290.003} C_VEL
LIN {X 0,Y 296.7,Z 548.824,A -85,B 0,C 180,E1 -16291.36,E2 -16291.36} C_VEL
LIN {X 0,Y 296.687,Z 547.098,A -85,B 0,C 180,E1 -16294.078,E2 -16294.078} C_VEL
LIN {X 0,Y 296.74,Z 544.984,A -85,B 0,C 180,E1 -16295.882,E2 -16295.882} C_VEL
LIN {X 0,Y 296.966,Z 541.224,A -85,B 0,C 180,E1 -16298.166,E2 -16298.166} C_VEL
LIN {X 0,Y 297.46,Z 536.693,A -85,B 0,C 180,E1 -16300.209,E2 -16300.209} C_VEL
LIN {X 0,Y 298.347,Z 529.816,A -85,B 0,C 180,E1 -16302.588,E2 -16302.588} C_VEL
LIN {X 0,Y 299.515,Z 522.355,A -85,B 0,C 180,E1 -16304.613,E2 -16304.613} C_VEL
LIN {X 0,Y 300.92,Z 513.397,A -85,B 0,C 180,E1 -16306.563,E2 -16306.563} C_VEL
LIN {X 0,Y 302.328,Z 503.427,A -85,B 0,C 180,E1 -16308.292,E2 -16308.292} C_VEL
LIN {X 0,Y 303.959,Z 492.764,A -85,B 0,C 180,E1 -16309.767,E2 -16309.767} C_VEL
LIN {X 0,Y 304.379,Z 488.583,A -85,B 0,C 180,E1 -16310.266,E2 -16310.266} C_VEL
LIN {X 0,Y 303.624,Z 476.754,A -85,B 0,C 180,E1 -16311.582,E2 -16311.582} C_VEL
LIN {X 0,Y 302.346,Z 464.252,A -85,B 0,C 180,E1 -16312.692,E2 -16312.692} C_VEL
LIN {X 0,Y 300.194,Z 450.895,A -85,B 0,C 180,E1 -16313.639,E2 -16313.639} C_VEL
LIN {X 0,Y 298.318,Z 441.4,A -85,B 0,C 180,E1 -16314.199,E2 -16314.199} C_VEL
LIN {X 0,Y 299.108,Z 434.944,A -85,B 0,C 180,E1 -16318.032,E2 -16318.032} C_VEL
LIN {X 0,Y 299.999,Z 428.727,A -85,B 0,C 180,E1 -16321.812,E2 -16321.812} C_VEL
LIN {X 0,Y 301.105,Z 422.514,A -85,B 0,C 180,E1 -16325.701,E2 -16325.701} C_VEL
LIN {X 0,Y 301.13,Z 418.718,A -85,B 0,C 180,E1 -16328.228,E2 -16328.228} C_VEL
LIN {X 0,Y 300.372,Z 414.088,A -85,B 0,C 180,E1 -16331.52,E2 -16331.52} C_VEL
LIN {X 0,Y 299.502,Z 409.137,A -85,B 0,C 180,E1 -16335.253,E2 -16335.253} C_VEL
LIN {X 0,Y 298.499,Z 403.726,A -85,B 0,C 180,E1 -16339.683,E2 -16339.683} C_VEL
LIN {X 0,Y 298.413,Z 403.314,A -85,B 0,C 180,E1 -16340.093,E2 -16340.093} C_VEL
LIN {X 0,Y 298.426,Z 403.311,A -85,B 0,C 180,E1 -16343.931,E2 -16343.931} C_VEL
LIN {X 0,Y 298.401,Z 403.314,A -85,B 0,C 180,E1 -16347.985,E2 -16347.985} C_VEL
LIN {X 0,Y 298.465,Z 403.306,A -85,B 0,C 180,E1 -16351.904,E2 -16351.904} C_VEL
LIN {X 0,Y 298.491,Z 403.304,A -85,B 0,C 180,E1 -16354.924,E2 -16354.924} C_VEL
LIN {X 0,Y 298.457,Z 403.307,A -85,B 0,C 180,E1 -16359.316,E2 -16359.316} C_VEL
LIN {X 0,Y 298.545,Z 403.299,A -85,B 0,C 180,E1 -16362.18,E2 -16362.18} C_VEL
LIN {X 0,Y 298.601,Z 403.29,A -85,B 0,C 180,E1 -16364.995,E2 -16364.995} C_VEL
LIN {X 0,Y 298.599,Z 403.289,A -85,B 0,C 180,E1 -16369.147,E2 -16369.147} C_VEL
LIN {X 0,Y 298.748,Z 403.272,A -85,B 0,C 180,E1 -16371.886,E2 -16371.886} C_VEL
LIN {X 0,Y 298.662,Z 403.282,A -85,B 0,C 180,E1 -16374.599,E2 -16374.599} C_VEL
LIN {X 0,Y 298.928,Z 403.247,A -85,B 0,C 180,E1 -16378.653,E2 -16378.653} C_VEL
LIN {X 0,Y 298.928,Z 403.247,A -85,B 0,C 180,E1 -16381.347,E2 -16381.347} C_VEL
LIN {X 0,Y 298.804,Z 403.253,A -85,B 0,C 180,E1 -16386.754,E2 -16386.754} C_VEL
LIN {X 0,Y 298.688,Z 403.273,A -85,B 0,C 180,E1 -16389.48,E2 -16389.48} C_VEL
LIN {X 0,Y 298.559,Z 403.296,A -85,B 0,C 180,E1 -16393.615,E2 -16393.615} C_VEL
LIN {X 0,Y 298.556,Z 403.291,A -85,B 0,C 180,E1 -16396.408,E2 -16396.408} C_VEL
LIN {X 0,Y 298.519,Z 403.293,A -85,B 0,C 180,E1 -16399.654,E2 -16399.654} C_VEL
LIN {X 0,Y 298.465,Z 403.306,A -85,B 0,C 180,E1 -16403.597,E2 -16403.597} C_VEL
LIN {X 0,Y 298.494,Z 403.301,A -85,B 0,C 180,E1 -16406.574,E2 -16406.574} C_VEL
LIN {X 0,Y 298.423,Z 403.31,A -85,B 0,C 180,E1 -16409.641,E2 -16409.641} C_VEL
LIN {X 0,Y 298.402,Z 403.305,A -85,B 0,C 180,E1 -16412.799,E2 -16412.799} C_VEL
LIN {X 0,Y 298.451,Z 403.306,A -85,B 0,C 180,E1 -16416.806,E2 -16416.806} C_VEL
LIN {X 0,Y 298.395,Z 403.316,A -85,B 0,C 180,E1 -16421.087,E2 -16421.087} C_VEL
LIN {X 0,Y 298.395,Z 403.312,A -85,B 0,C 180,E1 -16425.04,E2 -16425.04} C_VEL
LIN {X 0,Y 298.394,Z 403.316,A -85,B 0,C 180,E1 -16428.911,E2 -16428.911} C_VEL
LIN {X 0,Y 298.45,Z 403.308,A -85,B 0,C 180,E1 -16433.192,E2 -16433.192} C_VEL
LIN {X 0,Y 298.401,Z 403.316,A -85,B 0,C 180,E1 -16437.198,E2 -16437.198} C_VEL
LIN {X 0,Y 298.433,Z 403.309,A -85,B 0,C 180,E1 -16440.615,E2 -16440.615} C_VEL
LIN {X 0,Y 298.482,Z 403.305,A -85,B 0,C 180,E1 -16443.475,E2 -16443.475} C_VEL
LIN {X 0,Y 298.441,Z 403.31,A -85,B 0,C 180,E1 -16446.695,E2 -16446.695} C_VEL
LIN {X 0,Y 298.544,Z 403.297,A -85,B 0,C 180,E1 -16450.755,E2 -16450.755} C_VEL
LIN {X 0,Y 298.596,Z 403.291,A -85,B 0,C 180,E1 -16454.993,E2 -16454.993} C_VEL
LIN {X 0,Y 298.366,Z 403.319,A -85,B 0,C 180,E1 -16459.136,E2 -16459.136} C_VEL
LIN {X 0,Y 298.214,Z 403.667,A -85,B 0,C 180,E1 -16461.869,E2 -16461.869} C_VEL
LIN {X 0,Y 298.245,Z 405.784,A -85,B 0,C 180,E1 -16464.589,E2 -16464.589} C_VEL
LIN {X 0,Y 297.61,Z 409.711,A -85,B 0,C 180,E1 -16469.025,E2 -16469.025} C_VEL
LIN {X 0,Y 301.697,Z 422.941,A -85,B 0,C 180,E1 -16469.997,E2 -16469.997} C_VEL
LIN {X 0,Y 304.284,Z 432.126,A -85,B 0,C 180,E1 -16470.825,E2 -16470.825} C_VEL
LIN {X 0,Y 306.649,Z 443.799,A -85,B 0,C 180,E1 -16472.035,E2 -16472.035} C_VEL
LIN {X 0,Y 305.382,Z 455.649,A -85,B 0,C 180,E1 -16473.296,E2 -16473.296} C_VEL
LIN {X 0,Y 303.906,Z 466.77,A -85,B 0,C 180,E1 -16474.814,E2 -16474.814} C_VEL
LIN {X 0,Y 302.534,Z 475.771,A -85,B 0,C 180,E1 -16476.332,E2 -16476.332} C_VEL
LIN {X 0,Y 301.181,Z 484.078,A -85,B 0,C 180,E1 -16478.046,E2 -16478.046} C_VEL
LIN {X 0,Y 299.855,Z 492.221,A -85,B 0,C 180,E1 -16480.135,E2 -16480.135} C_VEL
LIN {X 0,Y 298.824,Z 498.613,A -85,B 0,C 180,E1 -16482.217,E2 -16482.217} C_VEL
LIN {X 0,Y 298.056,Z 503.389,A -85,B 0,C 180,E1 -16484.178,E2 -16484.178} C_VEL
LIN {X 0,Y 297.412,Z 507.633,A -85,B 0,C 180,E1 -16486.47,E2 -16486.47} C_VEL
LIN {X 0,Y 296.958,Z 510.636,A -85,B 0,C 180,E1 -16488.797,E2 -16488.797} C_VEL
